LIN {X 0,Y 282.338,Z 475.159,A -85,B 0,C 180,E1 -17007.146,E2 -17007.146} C_VEL
LIN {X 0,Y 282.332,Z 475.749,A -85,B 0,C 180,E1 -17008.574,E2 -17008.574} C_VEL
LIN {X 0,Y 282.332,Z 475.749,A -85,B 0,C 180,E1 -17011.426,E2 -17011.426} C_VEL
LIN {X 0,Y 282.337,Z 475.159,A -85,B 0,C 180,E1 -17012.854,E2 -17012.854} C_VEL
LIN {X 0,Y 282.387,Z 472.707,A -85,B 0,C 180,E1 -17015.713,E2 -17015.713} C_VEL
LIN {X 0,Y 282.677,Z 469.756,A -85,B 0,C 180,E1 -17017.859,E2 -17017.859} C_VEL
LIN {X 0,Y 283.174,Z 465.765,A -85,B 0,C 180,E1 -17020.005,E2 -17020.005} C_VEL
LIN {X 0,Y 283.966,Z 460.633,A -85,B 0,C 180,E1 -17022.144,E2 -17022.144} C_VEL
LIN {X 0,Y 284.95,Z 455.372,A -85,B 0,C 180,E1 -17023.914,E2 -17023.914} C_VEL
LIN {X 0,Y 286.08,Z 449.054,A -85,B 0,C 180,E1 -17025.678,E2 -17025.678} C_VEL
LIN {X 0,Y 287.263,Z 443.105,A -85,B 0,C 180,E1 -17027.073,E2 -17027.073} C_VEL
LIN {X 0,Y 288.401,Z 436.176,A -85,B 0,C 180,E1 -17028.469,E2 -17028.469} C_VEL
LIN {X 0,Y 289.842,Z 427.998,A -85,B 0,C 180,E1 -17029.844,E2 -17029.844} C_VEL
LIN {X 0,Y 291.314,Z 419.49,A -85,B 0,C 180,E1 -17031.03,E2 -17031.03} C_VEL
LIN {X 0,Y 292.62,Z 410.776,A -85,B 0,C 180,E1 -17032.041,E2 -17032.041} C_VEL
LIN {X 0,Y 293.928,Z 401.019,A -85,B 0,C 180,E1 -17032.957,E2 -17032.957} C_VEL
LIN {X 0,Y 295.008,Z 392.229,A -85,B 0,C 180,E1 -17033.611,E2 -17033.611} C_VEL
LIN {X 0,Y 295.879,Z 382.301,A -85,B 0,C 180,E1 -17034.188,E2 -17034.188} C_VEL
LIN {X 0,Y 296.551,Z 372.446,A -85,B 0,C 180,E1 -17034.596,E2 -17034.596} C_VEL
LIN {X 0,Y 297.291,Z 349.624,A -85,B 0,C 180,E1 -17035.184,E2 -17035.184} C_VEL
LIN {X 0,Y 298.183,Z 310.979,A -85,B 0,C 180,E1 -17036.113,E2 -17036.113} C_VEL
LIN {X 0,Y 294.142,Z 288.421,A -85,B 0,C 180,E1 -17037.1,E2 -17037.1} C_VEL
LIN {X 0,Y 290.092,Z 270.616,A -85,B 0,C 180,E1 -17037.994,E2 -17037.994} C_VEL
LIN {X 0,Y 288.061,Z 265.087,A -85,B 0,C 180,E1 -17038.405,E2 -17038.405} C_VEL
LIN {X 0,Y 287.295,Z 260.874,A -85,B 0,C 180,E1 -17040.098,E2 -17040.098} C_VEL
LIN {X 0,Y 285.623,Z 252.564,A -85,B 0,C 180,E1 -17043.784,E2 -17043.784} C_VEL
LIN {X 0,Y 284.361,Z 246.567,A -85,B 0,C 180,E1 -17046.602,E2 -17046.602} C_VEL
LIN {X 0,Y 284.308,Z 246.54,A -85,B 0,C 180,E1 -17049.994,E2 -17049.994} C_VEL
LIN {X 0,Y 284.248,Z 246.575,A -85,B 0,C 180,E1 -17054.19,E2 -17054.19} C_VEL
LIN {X 0,Y 284.274,Z 246.573,A -85,B 0,C 180,E1 -17058.124,E2 -17058.124} C_VEL
LIN {X 0,Y 284.328,Z 246.568,A -85,B 0,C 180,E1 -17062.276,E2 -17062.276} C_VEL
LIN {X 0,Y 284.31,Z 246.548,A -85,B 0,C 180,E1 -17065.35,E2 -17065.35} C_VEL
LIN {X 0,Y 284.295,Z 246.57,A -85,B 0,C 180,E1 -17068.725,E2 -17068.725} C_VEL
LIN {X 0,Y 284.393,Z 246.531,A -85,B 0,C 180,E1 -17072.828,E2 -17072.828} C_VEL
LIN {X 0,Y 284.367,Z 246.56,A -85,B 0,C 180,E1 -17076.706,E2 -17076.706} C_VEL
LIN {X 0,Y 284.383,Z 246.524,A -85,B 0,C 180,E1 -17081.259,E2 -17081.259} C_VEL
LIN {X 0,Y 284.468,Z 246.547,A -85,B 0,C 180,E1 -17085.696,E2 -17085.696} C_VEL
LIN {X 0,Y 284.514,Z 246.504,A -85,B 0,C 180,E1 -17090.042,E2 -17090.042} C_VEL
LIN {X 0,Y 284.653,Z 246.511,A -85,B 0,C 180,E1 -17092.908,E2 -17092.908} C_VEL
LIN {X 0,Y 284.741,Z 246.506,A -85,B 0,C 180,E1 -17097.17,E2 -17097.17} C_VEL
LIN {X 0,Y 284.911,Z 246.454,A -85,B 0,C 180,E1 -17099.999,E2 -17099.999} C_VEL
LIN {X 0,Y 284.743,Z 246.501,A -85,B 0,C 180,E1 -17102.829,E2 -17102.829} C_VEL
LIN {X 0,Y 284.685,Z 246.512,A -85,B 0,C 180,E1 -17107.09,E2 -17107.09} C_VEL
LIN {X 0,Y 284.518,Z 246.504,A -85,B 0,C 180,E1 -17109.956,E2 -17109.956} C_VEL
LIN {X 0,Y 284.48,Z 246.549,A -85,B 0,C 180,E1 -17114.302,E2 -17114.302} C_VEL
LIN {X 0,Y 284.421,Z 246.539,A -85,B 0,C 180,E1 -17117.248,E2 -17117.248} C_VEL
LIN {X 0,Y 284.375,Z 246.533,A -85,B 0,C 180,E1 -17120.242,E2 -17120.242} C_VEL
LIN {X 0,Y 284.334,Z 246.56,A -85,B 0,C 180,E1 -17124.846,E2 -17124.846} C_VEL
LIN {X 0,Y 284.324,Z 246.54,A -85,B 0,C 180,E1 -17128.01,E2 -17128.01} C_VEL
LIN {X 0,Y 284.293,Z 246.573,A -85,B 0,C 180,E1 -17131.274,E2 -17131.274} C_VEL
LIN {X 0,Y 284.359,Z 246.546,A -85,B 0,C 180,E1 -17135.353,E2 -17135.353} C_VEL
LIN {X 0,Y 284.333,Z 246.568,A -85,B 0,C 180,E1 -17138.165,E2 -17138.165} C_VEL
LIN {X 0,Y 284.338,Z 246.558,A -85,B 0,C 180,E1 -17142.14,E2 -17142.14} C_VEL
LIN {X 0,Y 284.293,Z 246.533,A -85,B 0,C 180,E1 -17146.197,E2 -17146.197} C_VEL
LIN {X 0,Y 284.309,Z 246.538,A -85,B 0,C 180,E1 -17150.022,E2 -17150.022} C_VEL
LIN {X 0,Y 284.349,Z 246.546,A -85,B 0,C 180,E1 -17153.617,E2 -17153.617} C_VEL
LIN {X 0,Y 284.304,Z 246.553,A -85,B 0,C 180,E1 -17157.189,E2 -17157.189} C_VEL
LIN {X 0,Y 284.357,Z 246.706,A -85,B 0,C 180,E1 -17160.852,E2 -17160.852} C_VEL
LIN {X 0,Y 284.57,Z 247.628,A -85,B 0,C 180,E1 -17161.125,E2 -17161.125} C_VEL
LIN {X 0,Y 292.692,Z 262.865,A -85,B 0,C 180,E1 -17162.446,E2 -17162.446} C_VEL
LIN {X 0,Y 300.724,Z 274.196,A -85,B 0,C 180,E1 -17163.545,E2 -17163.545} C_VEL
LIN {X 0,Y 308.771,Z 283.256,A -85,B 0,C 180,E1 -17164.599,E2 -17164.599} C_VEL
LIN {X 0,Y 316.781,Z 291.82,A -85,B 0,C 180,E1 -17165.796,E2 -17165.796} C_VEL
LIN {X 0,Y 324.604,Z 299.651,A -85,B 0,C 180,E1 -17167.139,E2 -17167.139} C_VEL
LIN {X 0,Y 333.028,Z 307.638,A -85,B 0,C 180,E1 -17168.762,E2 -17168.762} C_VEL
LIN {X 0,Y 340.838,Z 314.592,A -85,B 0,C 180,E1 -17170.439,E2 -17170.439} C_VEL
LIN {X 0,Y 346.811,Z 319.308,A -85,B 0,C 180,E1 -17171.823,E2 -17171.823} C_VEL
LIN {X 0,Y 352.868,Z 324.611,A -85,B 0,C 180,E1 -17173.385,E2 -17173.385} C_VEL
LIN {X 0,Y 358.666,Z 328.923,A -85,B 0,C 180,E1 -17175.022,E2 -17175.022} C_VEL
LIN {X 0,Y 363.783,Z 333.09,A -85,B 0,C 180,E1 -17176.663,E2 -17176.663} C_VEL
LIN {X 0,Y 368.41,Z 336.029,A -85,B 0,C 180,E1 -17178.317,E2 -17178.317} C_VEL
LIN {X 0,Y 370.505,Z 337.411,A -85,B 0,C 180,E1 -17179.169,E2 -17179.169} C_VEL
LIN {X 0,Y 373.81,Z 340.321,A -85,B 0,C 180,E1 -17180.705,E2 -17180.705} C_VEL
LIN {X 0,Y 376.908,Z 342.491,A -85,B 0,C 180,E1 -17182.387,E2 -17182.387} C_VEL
LIN {X 0,Y 379.747,Z 344.052,A -85,B 0,C 180,E1 -17184.313,E2 -17184.313} C_VEL
LIN {X 0,Y 381.691,Z 344.805,A -85,B 0,C 180,E1 -17186.15,E2 -17186.15} C_VEL
LIN {X 0,Y 382.967,Z 345.365,A -85,B 0,C 180,E1 -17188.16,E2 -17188.16} C_VEL
LIN {X 0,Y 383.351,Z 345.508,A -85,B 0,C 180,E1 -17190,E2 -17190} C_VEL
LIN {X 0,Y 383.05,Z 345.431,A -85,B 0,C 180,E1 -17191.577,E2 -17191.577} C_VEL
LIN {X 0,Y 382.23,Z 344.938,A -85,B 0,C 180,E1 -17193.162,E2 -17193.162} C_VEL
LIN {X 0,Y 380.501,Z 344.425,A -85,B 0,C 180,E1 -17195.024,E2 -17195.024} C_VEL
LIN {X 0,Y 377.946,Z 343.114,A -85,B 0,C 180,E1 -17196.961,E2 -17196.961} C_VEL
LIN {X 0,Y 374.623,Z 340.95,A -85,B 0,C 180,E1 -17198.885,E2 -17198.885} C_VEL
LIN {X 0,Y 371.033,Z 337.887,A -85,B 0,C 180,E1 -17200.604,E2 -17200.604} C_VEL
LIN {X 0,Y 368.789,Z 336.215,A -85,B 0,C 180,E1 -17201.535,E2 -17201.535} C_VEL
LIN {X 0,Y 364.035,Z 333.254,A -85,B 0,C 180,E1 -17203.255,E2 -17203.255} C_VEL
LIN {X 0,Y 359.028,Z 329.244,A -85,B 0,C 180,E1 -17204.863,E2 -17204.863} C_VEL
LIN {X 0,Y 354.264,Z 325.619,A -85,B 0,C 180,E1 -17206.237,E2 -17206.237} C_VEL
LIN {X 0,Y 348.703,Z 321.024,A -85,B 0,C 180,E1 -17207.707,E2 -17207.707} C_VEL
LIN {X 0,Y 341.134,Z 314.874,A -85,B 0,C 180,E1 -17209.492,E2 -17209.492} C_VEL
LIN {X 0,Y 335.412,Z 309.793,A -85,B 0,C 180,E1 -17210.737,E2 -17210.737} C_VEL
LIN {X 0,Y 329.61,Z 304.23,A -85,B 0,C 180,E1 -17211.926,E2 -17211.926} C_VEL
LIN {X 0,Y 323.047,Z 298.018,A -85,B 0,C 180,E1 -17213.151,E2 -17213.151} C_VEL
LIN {X 0,Y 316.393,Z 291.393,A -85,B 0,C 180,E1 -17214.263,E2 -17214.263} C_VEL
LIN {X 0,Y 308.203,Z 282.711,A -85,B 0,C 180,E1 -17215.475,E2 -17215.475} C_VEL
LIN {X 0,Y 299.727,Z 272.881,A -85,B 0,C 180,E1 -17216.585,E2 -17216.585} C_VEL
LIN {X 0,Y 292.26,Z 262.125,A -85,B 0,C 180,E1 -17217.619,E2 -17217.619} C_VEL
LIN {X 0,Y 284.572,Z 247.623,A -85,B 0,C 180,E1 -17218.876,E2 -17218.876} C_VEL
LIN {X 0,Y 284.349,Z 246.627,A -85,B 0,C 180,E1 -17219.19,E2 -17219.19} C_VEL
LIN {X 0,Y 284.302,Z 246.551,A -85,B 0,C 180,E1 -17222.946,E2 -17222.946} C_VEL
LIN {X 0,Y 284.349,Z 246.546,A -85,B 0,C 180,E1 -17226.383,E2 -17226.383} C_VEL
LIN {X 0,Y 284.308,Z 246.538,A -85,B 0,C 180,E1 -17229.994,E2 -17229.994} C_VEL
LIN {X 0,Y 284.29,Z 246.542,A -85,B 0,C 180,E1 -17234.201,E2 -17234.201} C_VEL
LIN {X 0,Y 284.336,Z 246.556,A -85,B 0,C 180,E1 -17238.137,E2 -17238.137} C_VEL
LIN {X 0,Y 284.342,Z 246.568,A -85,B 0,C 180,E1 -17242.272,E2 -17242.272} C_VEL
LIN {X 0,Y 284.321,Z 246.547,A -85,B 0,C 180,E1 -17245.353,E2 -17245.353} C_VEL
LIN {X 0,Y 284.293,Z 246.573,A -85,B 0,C 180,E1 -17248.726,E2 -17248.726} C_VEL
LIN {X 0,Y 284.39,Z 246.53,A -85,B 0,C 180,E1 -17252.829,E2 -17252.829} C_VEL
LIN {X 0,Y 284.331,Z 246.567,A -85,B 0,C 180,E1 -17256.705,E2 -17256.705} C_VEL
LIN {X 0,Y 284.397,Z 246.524,A -85,B 0,C 180,E1 -17261.262,E2 -17261.262} C_VEL
LIN {X 0,Y 284.491,Z 246.545,A -85,B 0,C 180,E1 -17264.46,E2 -17264.46} C_VEL
LIN {X 0,Y 284.486,Z 246.52,A -85,B 0,C 180,E1 -17268.602,E2 -17268.602} C_VEL
LIN {X 0,Y 284.638,Z 246.499,A -85,B 0,C 180,E1 -17271.481,E2 -17271.481} C_VEL
LIN {X 0,Y 284.596,Z 246.533,A -85,B 0,C 180,E1 -17274.332,E2 -17274.332} C_VEL
LIN {X 0,Y 284.854,Z 246.468,A -85,B 0,C 180,E1 -17278.587,E2 -17278.587} C_VEL
LIN {X 0,Y 284.854,Z 246.474,A -85,B 0,C 180,E1 -17281.415,E2 -17281.415} C_VEL
LIN {X 0,Y 284.581,Z 246.533,A -85,B 0,C 180,E1 -17285.67,E2 -17285.67} C_VEL
LIN {X 0,Y 284.615,Z 246.493,A -85,B 0,C 180,E1 -17288.99,E2 -17288.99} C_VEL
LIN {X 0,Y 284.473,Z 246.541,A -85,B 0,C 180,E1 -17292.848,E2 -17292.848} C_VEL
LIN {X 0,Y 284.427,Z 246.546,A -85,B 0,C 180,E1 -17295.772,E2 -17295.772} C_VEL
LIN {X 0,Y 284.383,Z 246.534,A -85,B 0,C 180,E1 -17299.999,E2 -17299.999} C_VEL
LIN {X 0,Y 283.755,Z 246.629,A -85,B 0,C 180,E1 -17301.182,E2 -17301.182} C_VEL
LIN {X 0,Y 280.878,Z 246.995,A -85,B 0,C 180,E1 -17303.107,E2 -17303.107} C_VEL
LIN {X 0,Y 278.419,Z 247.291,A -85,B 0,C 180,E1 -17304.672,E2 -17304.672} C_VEL
LIN {X 0,Y 277.379,Z 247.408,A -85,B 0,C 180,E1 -17305.885,E2 -17305.885} C_VEL
LIN {X 0,Y 277.305,Z 247.414,A -85,B 0,C 180,E1 -17306.296,E2 -17306.296} C_VEL
LIN {X 0,Y 277.273,Z 247.448,A -85,B 0,C 180,E1 -17310.482,E2 -17310.482} C_VEL
LIN {X 0,Y 277.248,Z 247.426,A -85,B 0,C 180,E1 -17313.896,E2 -17313.896} C_VEL
LIN {X 0,Y 277.273,Z 247.446,A -85,B 0,C 180,E1 -17317.469,E2 -17317.469} C_VEL
LIN {X 0,Y 277.212,Z 247.447,A -85,B 0,C 180,E1 -17321.237,E2 -17321.237} C_VEL
LIN {X 0,Y 277.203,Z 247.448,A -85,B 0,C 180,E1 -17325.227,E2 -17325.227} C_VEL
LIN {X 0,Y 277.224,Z 247.421,A -85,B 0,C 180,E1 -17329.513,E2 -17329.513} C_VEL
LIN {X 0,Y 277.351,Z 247.644,A -85,B 0,C 180,E1 -17332.961,E2 -17332.961} C_VEL
LIN {X 0,Y 278.847,Z 254.731,A -85,B 0,C 180,E1 -17336.325,E2 -17336.325} C_VEL
LIN {X 0,Y 280.431,Z 262.591,A -85,B 0,C 180,E1 -17339.919,E2 -17339.919} C_VEL
LIN {X 0,Y 280.834,Z 264.832,A -85,B 0,C 180,E1 -17340.786,E2 -17340.786} C_VEL
LIN {X 0,Y 284.402,Z 274.054,A -85,B 0,C 180,E1 -17341.497,E2 -17341.497} C_VEL
LIN {X 0,Y 289.1,Z 296.203,A -85,B 0,C 180,E1 -17342.605,E2 -17342.605} C_VEL
LIN {X 0,Y 291.885,Z 312.955,A -85,B 0,C 180,E1 -17343.338,E2 -17343.338} C_VEL
LIN {X 0,Y 290.193,Z 370.926,A -85,B 0,C 180,E1 -17344.78,E2 -17344.78} C_VEL
LIN {X 0,Y 289.497,Z 381.234,A -85,B 0,C 180,E1 -17345.195,E2 -17345.195} C_VEL
LIN {X 0,Y 288.564,Z 390.746,A -85,B 0,C 180,E1 -17345.733,E2 -17345.733} C_VEL
LIN {X 0,Y 287.493,Z 399.819,A -85,B 0,C 180,E1 -17346.403,E2 -17346.403} C_VEL
LIN {X 0,Y 286.24,Z 408.95,A -85,B 0,C 180,E1 -17347.25,E2 -17347.25} C_VEL
LIN {X 0,Y 284.929,Z 417.946,A -85,B 0,C 180,E1 -17348.285,E2 -17348.285} C_VEL
LIN {X 0,Y 283.358,Z 426.67,A -85,B 0,C 180,E1 -17349.492,E2 -17349.492} C_VEL
LIN {X 0,Y 281.981,Z 434.062,A -85,B 0,C 180,E1 -17350.717,E2 -17350.717} C_VEL
LIN {X 0,Y 280.72,Z 441.747,A -85,B 0,C 180,E1 -17352.247,E2 -17352.247} C_VEL
LIN {X 0,Y 279.228,Z 448.861,A -85,B 0,C 180,E1 -17353.927,E2 -17353.927} C_VEL
LIN {X 0,Y 278.016,Z 455.178,A -85,B 0,C 180,E1 -17355.731,E2 -17355.731} C_VEL
LIN {X 0,Y 276.987,Z 460.439,A -85,B 0,C 180,E1 -17357.545,E2 -17357.545} C_VEL
LIN {X 0,Y 276.165,Z 465.572,A -85,B 0,C 180,E1 -17359.739,E2 -17359.739} C_VEL
LIN {X 0,Y 275.606,Z 469.562,A -85,B 0,C 180,E1 -17361.938,E2 -17361.938} C_VEL
LIN {X 0,Y 275.254,Z 473.199,A -85,B 0,C 180,E1 -17364.741,E2 -17364.741} C_VEL
LIN {X 0,Y 275.247,Z 474.966,A -85,B 0,C 180,E1 -17367.073,E2 -17367.073} C_VEL
LIN {X 0,Y 275.256,Z 475.557,A -85,B 0,C 180,E1 -17368.537,E2 -17368.537} C_VEL
LIN {X 0,Y 275.256,Z 475.557,A -85,B 0,C 180,E1 -17371.463,E2 -17371.463} C_VEL
LIN {X 0,Y 275.246,Z 474.966,A -85,B 0,C 180,E1 -17372.927,E2 -17372.927} C_VEL
LIN {X 0,Y 275.3,Z 472.514,A -85,B 0,C 180,E1 -17375.861,E2 -17375.861} C_VEL
LIN {X 0,Y 275.606,Z 469.562,A -85,B 0,C 180,E1 -17378.062,E2 -17378.062} C_VEL
LIN {X 0,Y 276.165,Z 465.572,A -85,B 0,C 180,E1 -17380.261,E2 -17380.261} C_VEL
LIN {X 0,Y 276.987,Z 460.439,A -85,B 0,C 180,E1 -17382.455,E2 -17382.455} C_VEL
LIN {X 0,Y 278.014,Z 455.178,A -85,B 0,C 180,E1 -17384.269,E2 -17384.269} C_VEL
LIN {X 0,Y 279.217,Z 448.86,A -85,B 0,C 180,E1 -17386.074,E2 -17386.074} C_VEL
LIN {X 0,Y 280.666,Z 441.91,A -85,B 0,C 180,E1 -17387.718,E2 -17387.718} C_VEL
LIN {X 0,Y 281.662,Z 435.982,A -85,B 0,C 180,E1 -17388.928,E2 -17388.928} C_VEL
LIN {X 0,Y 283.168,Z 427.805,A -85,B 0,C 180,E1 -17390.332,E2 -17390.332} C_VEL
LIN {X 0,Y 284.696,Z 419.297,A -85,B 0,C 180,E1 -17391.543,E2 -17391.543} C_VEL
LIN {X 0,Y 286.054,Z 410.583,A -85,B 0,C 180,E1 -17392.575,E2 -17392.575} C_VEL
LIN {X 0,Y 287.275,Z 401.833,A -85,B 0,C 180,E1 -17393.425,E2 -17393.425} C_VEL
LIN {X 0,Y 288.514,Z 392.036,A -85,B 0,C 180,E1 -17394.176,E2 -17394.176} C_VEL
LIN {X 0,Y 289.425,Z 382.108,A -85,B 0,C 180,E1 -17394.763,E2 -17394.763} C_VEL
LIN {X 0,Y 290.129,Z 372.254,A -85,B 0,C 180,E1 -17395.178,E2 -17395.178} C_VEL
LIN {X 0,Y 290.87,Z 349.431,A -85,B 0,C 180,E1 -17395.78,E2 -17395.78} C_VEL
LIN {X 0,Y 291.736,Z 311.475,A -85,B 0,C 180,E1 -17396.717,E2 -17396.717} C_VEL
LIN {X 0,Y 288.006,Z 290.521,A -85,B 0,C 180,E1 -17397.663,E2 -17397.663} C_VEL
LIN {X 0,Y 284.029,Z 272.943,A -85,B 0,C 180,E1 -17398.575,E2 -17398.575} C_VEL
LIN {X 0,Y 280.833,Z 264.881,A -85,B 0,C 180,E1 -17399.205,E2 -17399.205} C_VEL
LIN {X 0,Y 280.133,Z 261.18,A -85,B 0,C 180,E1 -17400.726,E2 -17400.726} C_VEL
LIN {X 0,Y 278.413,Z 252.737,A -85,B 0,C 180,E1 -17404.608,E2 -17404.608} C_VEL
LIN {X 0,Y 277.328,Z 247.446,A -85,B 0,C 180,E1 -17407.198,E2 -17407.198} C_VEL
LIN {X 0,Y 277.212,Z 247.425,A -85,B 0,C 180,E1 -17411.236,E2 -17411.236} C_VEL
LIN {X 0,Y 277.203,Z 247.445,A -85,B 0,C 180,E1 -17415.226,E2 -17415.226} C_VEL
LIN {X 0,Y 277.224,Z 247.438,A -85,B 0,C 180,E1 -17419.511,E2 -17419.511} C_VEL
LIN {X 0,Y 277.273,Z 247.446,A -85,B 0,C 180,E1 -17422.531,E2 -17422.531} C_VEL
LIN {X 0,Y 277.248,Z 247.426,A -85,B 0,C 180,E1 -17426.104,E2 -17426.104} C_VEL
LIN {X 0,Y 277.263,Z 247.449,A -85,B 0,C 180,E1 -17429.538,E2 -17429.538} C_VEL
LIN {X 0,Y 277.355,Z 247.407,A -85,B 0,C 180,E1 -17432.863,E2 -17432.863} C_VEL
LIN {X 0,Y 277.329,Z 247.436,A -85,B 0,C 180,E1 -17436.079,E2 -17436.079} C_VEL
LIN {X 0,Y 277.333,Z 247.403,A -85,B 0,C 180,E1 -17440.765,E2 -17440.765} C_VEL
LIN {X 0,Y 277.415,Z 247.427,A -85,B 0,C 180,E1 -17445.324,E2 -17445.324} C_VEL
LIN {X 0,Y 277.457,Z 247.384,A -85,B 0,C 180,E1 -17449.786,E2 -17449.786} C_VEL
LIN {X 0,Y 277.611,Z 247.386,A -85,B 0,C 180,E1 -17452.727,E2 -17452.727} C_VEL
LIN {X 0,Y 277.82,Z 247.35,A -85,B 0,C 180,E1 -17458.55,E2 -17458.55} C_VEL
LIN {X 0,Y 277.82,Z 247.344,A -85,B 0,C 180,E1 -17461.449,E2 -17461.449} C_VEL
LIN {X 0,Y 277.64,Z 247.389,A -85,B 0,C 180,E1 -17467.27,E2 -17467.27} C_VEL
LIN {X 0,Y 277.46,Z 247.383,A -85,B 0,C 180,E1 -17470.212,E2 -17470.212} C_VEL
LIN {X 0,Y 277.433,Z 247.428,A -85,B 0,C 180,E1 -17474.673,E2 -17474.673} C_VEL
LIN {X 0,Y 277.34,Z 247.402,A -85,B 0,C 180,E1 -17479.233,E2 -17479.233} C_VEL
LIN {X 0,Y 277.289,Z 247.444,A -85,B 0,C 180,E1 -17484.157,E2 -17484.157} C_VEL
LIN {X 0,Y 277.319,Z 247.41,A -85,B 0,C 180,E1 -17487.503,E2 -17487.503} C_VEL
LIN {X 0,Y 277.269,Z 247.448,A -85,B 0,C 180,E1 -17490.481,E2 -17490.481} C_VEL
LIN {X 0,Y 277.251,Z 247.429,A -85,B 0,C 180,E1 -17493.894,E2 -17493.894} C_VEL
LIN {X 0,Y 277.287,Z 247.446,A -85,B 0,C 180,E1 -17497.465,E2 -17497.465} C_VEL
LIN {X 0,Y 277.261,Z 247.431,A -85,B 0,C 180,E1 -17501.226,E2 -17501.226} C_VEL
LIN {X 0,Y 277.239,Z 247.431,A -85,B 0,C 180,E1 -17505.217,E2 -17505.217} C_VEL
LIN {X 0,Y 277.225,Z 247.408,A -85,B 0,C 180,E1 -17509.51,E2 -17509.51} C_VEL
LIN {X 0,Y 277.285,Z 247.446,A -85,B 0,C 180,E1 -17512.534,E2 -17512.534} C_VEL
LIN {X 0,Y 277.25,Z 247.416,A -85,B 0,C 180,E1 -17516.105,E2 -17516.105} C_VEL
LIN {X 0,Y 277.306,Z 247.573,A -85,B 0,C 180,E1 -17520.072,E2 -17520.072} C_VEL
LIN {X 0,Y 277.558,Z 248.55,A -85,B 0,C 180,E1 -17520.348,E2 -17520.348} C_VEL
LIN {X 0,Y 287.678,Z 267.474,A -85,B 0,C 180,E1 -17522.047,E2 -17522.047} C_VEL
LIN {X 0,Y 296.035,Z 279.257,A -85,B 0,C 180,E1 -17523.224,E2 -17523.224} C_VEL
LIN {X 0,Y 304.941,Z 289.145,A -85,B 0,C 180,E1 -17524.349,E2 -17524.349} C_VEL
LIN {X 0,Y 313.119,Z 297.715,A -85,B 0,C 180,E1 -17525.493,E2 -17525.493} C_VEL
LIN {X 0,Y 322.054,Z 306.384,A -85,B 0,C 180,E1 -17526.937,E2 -17526.937} C_VEL
LIN {X 0,Y 330.86,Z 314.506,A -85,B 0,C 180,E1 -17528.59,E2 -17528.59} C_VEL
LIN {X 0,Y 339.989,Z 322.423,A -85,B 0,C 180,E1 -17530.519,E2 -17530.519} C_VEL
LIN {X 0,Y 346.429,Z 327.558,A -85,B 0,C 180,E1 -17532.016,E2 -17532.016} C_VEL
LIN {X 0,Y 352.732,Z 332.614,A -85,B 0,C 180,E1 -17533.635,E2 -17533.635} C_VEL
LIN {X 0,Y 356.978,Z 335.771,A -85,B 0,C 180,E1 -17534.83,E2 -17534.83} C_VEL
LIN {X 0,Y 362.424,Z 340.053,A -85,B 0,C 180,E1 -17536.544,E2 -17536.544} C_VEL
LIN {X 0,Y 367.359,Z 343.081,A -85,B 0,C 180,E1 -17538.284,E2 -17538.284} C_VEL
LIN {X 0,Y 369.339,Z 344.533,A -85,B 0,C 180,E1 -17539.082,E2 -17539.082} C_VEL
LIN {X 0,Y 373.007,Z 347.551,A -85,B 0,C 180,E1 -17540.763,E2 -17540.763} C_VEL
LIN {X 0,Y 376.178,Z 349.68,A -85,B 0,C 180,E1 -17542.485,E2 -17542.485} C_VEL
LIN {X 0,Y 378.846,Z 351.099,A -85,B 0,C 180,E1 -17544.3,E2 -17544.3} C_VEL
LIN {X 0,Y 380.516,Z 351.761,A -85,B 0,C 180,E1 -17545.826,E2 -17545.826} C_VEL
LIN {X 0,Y 381.686,Z 352.195,A -85,B 0,C 180,E1 -17547.349,E2 -17547.349} C_VEL
LIN {X 0,Y 382.346,Z 352.596,A -85,B 0,C 180,E1 -17548.947,E2 -17548.947} C_VEL
LIN {X 0,Y 382.488,Z 352.539,A -85,B 0,C 180,E1 -17550,E2 -17550} C_VEL
LIN {X 0,Y 382.181,Z 352.479,A -85,B 0,C 180,E1 -17551.581,E2 -17551.581} C_VEL
LIN {X 0,Y 381.093,Z 351.917,A -85,B 0,C 180,E1 -17553.514,E2 -17553.514} C_VEL
LIN {X 0,Y 379.106,Z 351.218,A -85,B 0,C 180,E1 -17555.477,E2 -17555.477} C_VEL
LIN {X 0,Y 376.465,Z 349.809,A -85,B 0,C 180,E1 -17557.348,E2 -17557.348} C_VEL
LIN {X 0,Y 373.181,Z 347.677,A -85,B 0,C 180,E1 -17559.154,E2 -17559.154} C_VEL
LIN {X 0,Y 369.654,Z 344.778,A -85,B 0,C 180,E1 -17560.785,E2 -17560.785} C_VEL
LIN {X 0,Y 366.939,Z 342.836,A -85,B 0,C 180,E1 -17561.871,E2 -17561.871} C_VEL
LIN {X 0,Y 362.246,Z 339.915,A -85,B 0,C 180,E1 -17563.516,E2 -17563.516} C_VEL
LIN {X 0,Y 356.744,Z 335.561,A -85,B 0,C 180,E1 -17565.24,E2 -17565.24} C_VEL
LIN {X 0,Y 349.772,Z 330.397,A -85,B 0,C 180,E1 -17567.136,E2 -17567.136} C_VEL
LIN {X 0,Y 342.455,Z 324.339,A -85,B 0,C 180,E1 -17568.928,E2 -17568.928} C_VEL
LIN {X 0,Y 336.047,Z 318.959,A -85,B 0,C 180,E1 -17570.342,E2 -17570.342} C_VEL
LIN {X 0,Y 328.443,Z 312.315,A -85,B 0,C 180,E1 -17571.883,E2 -17571.883} C_VEL
LIN {X 0,Y 320.06,Z 304.416,A -85,B 0,C 180,E1 -17573.402,E2 -17573.402} C_VEL
LIN {X 0,Y 312.403,Z 296.949,A -85,B 0,C 180,E1 -17574.611,E2 -17574.611} C_VEL
LIN {X 0,Y 303.963,Z 288.179,A -85,B 0,C 180,E1 -17575.775,E2 -17575.775} C_VEL
LIN {X 0,Y 294.557,Z 277.321,A -85,B 0,C 180,E1 -17576.975,E2 -17576.975} C_VEL
LIN {X 0,Y 287.007,Z 266.35,A -85,B 0,C 180,E1 -17578.056,E2 -17578.056} C_VEL
LIN {X 0,Y 277.55,Z 248.559,A -85,B 0,C 180,E1 -17579.65,E2 -17579.65} C_VEL
LIN {X 0,Y 277.302,Z 247.519,A -85,B 0,C 180,E1 -17579.965,E2 -17579.965} C_VEL
LIN {X 0,Y 277.25,Z 247.416,A -85,B 0,C 180,E1 -17583.895,E2 -17583.895} C_VEL
LIN {X 0,Y 277.285,Z 247.446,A -85,B 0,C 180,E1 -17587.466,E2 -17587.466} C_VEL
LIN {X 0,Y 277.214,Z 247.401,A -85,B 0,C 180,E1 -17591.235,E2 -17591.235} C_VEL
LIN {X 0,Y 277.243,Z 247.439,A -85,B 0,C 180,E1 -17595.217,E2 -17595.217} C_VEL
LIN {X 0,Y 277.292,Z 247.426,A -85,B 0,C 180,E1 -17599.495,E2 -17599.495} C_VEL
LIN {X 0,Y 277.287,Z 247.446,A -85,B 0,C 180,E1 -17602.535,E2 -17602.535} C_VEL
LIN {X 0,Y 277.251,Z 247.429,A -85,B 0,C 180,E1 -17606.106,E2 -17606.106} C_VEL
LIN {X 0,Y 277.259,Z 247.449,A -85,B 0,C 180,E1 -17609.539,E2 -17609.539} C_VEL
LIN {X 0,Y 277.352,Z 247.406,A -85,B 0,C 180,E1 -17612.864,E2 -17612.864} C_VEL
LIN {X 0,Y 277.295,Z 247.445,A -85,B 0,C 180,E1 -17616.077,E2 -17616.077} C_VEL
LIN {X 0,Y 277.34,Z 247.402,A -85,B 0,C 180,E1 -17620.767,E2 -17620.767} C_VEL
LIN {X 0,Y 277.433,Z 247.428,A -85,B 0,C 180,E1 -17625.327,E2 -17625.327} C_VEL
LIN {X 0,Y 277.46,Z 247.383,A -85,B 0,C 180,E1 -17629.788,E2 -17629.788} C_VEL
LIN {X 0,Y 277.64,Z 247.389,A -85,B 0,C 180,E1 -17632.73,E2 -17632.73} C_VEL
LIN {X 0,Y 277.82,Z 247.344,A -85,B 0,C 180,E1 -17638.551,E2 -17638.551} C_VEL
LIN {X 0,Y 277.82,Z 247.35,A -85,B 0,C 180,E1 -17641.45,E2 -17641.45} C_VEL
LIN {X 0,Y 277.611,Z 247.386,A -85,B 0,C 180,E1 -17647.273,E2 -17647.273} C_VEL
LIN {X 0,Y 277.457,Z 247.384,A -85,B 0,C 180,E1 -17650.214,E2 -17650.214} C_VEL
LIN {X 0,Y 277.415,Z 247.427,A -85,B 0,C 180,E1 -17654.676,E2 -17654.676} C_VEL
LIN {X 0,Y 277.333,Z 247.403,A -85,B 0,C 180,E1 -17659.235,E2 -17659.235} C_VEL
LIN {X 0,Y 277.329,Z 247.436,A -85,B 0,C 180,E1 -17663.921,E2 -17663.921} C_VEL
LIN {X 0,Y 277.305,Z 247.414,A -85,B 0,C 180,E1 -17666.296,E2 -17666.296} C_VEL
LIN {X 0,Y 276.644,Z 247.5,A -85,B 0,C 180,E1 -17667.508,E2 -17667.508} C_VEL
LIN {X 0,Y 273.728,Z 247.885,A -85,B 0,C 180,E1 -17669.48,E2 -17669.48} C_VEL
LIN {X 0,Y 271.265,Z 248.194,A -85,B 0,C 180,E1 -17671.083,E2 -17671.083} C_VEL
LIN {X 0,Y 270.243,Z 248.311,A -85,B 0,C 180,E1 -17672.328,E2 -17672.328} C_VEL
LIN {X 0,Y 270.179,Z 248.312,A -85,B 0,C 180,E1 -17672.749,E2 -17672.749} C_VEL
LIN {X 0,Y 270.229,Z 248.323,A -85,B 0,C 180,E1 -17676.74,E2 -17676.74} C_VEL
LIN {X 0,Y 270.171,Z 248.321,A -85,B 0,C 180,E1 -17681.029,E2 -17681.029} C_VEL
LIN {X 0,Y 270.154,Z 248.327,A -85,B 0,C 180,E1 -17685.381,E2 -17685.381} C_VEL
LIN {X 0,Y 270.176,Z 248.298,A -85,B 0,C 180,E1 -17689.435,E2 -17689.435} C_VEL
LIN {X 0,Y 270.284,Z 248.51,A -85,B 0,C 180,E1 -17692.335,E2 -17692.335} C_VEL
LIN {X 0,Y 271.788,Z 255.647,A -85,B 0,C 180,E1 -17695.841,E2 -17695.841} C_VEL
LIN {X 0,Y 273.486,Z 264.006,A -85,B 0,C 180,E1 -17699.764,E2 -17699.764} C_VEL
LIN {X 0,Y 273.78,Z 265.178,A -85,B 0,C 180,E1 -17700.007,E2 -17700.007} C_VEL
LIN {X 0,Y 278.471,Z 276.628,A -85,B 0,C 180,E1 -17700.912,E2 -17700.912} C_VEL
LIN {X 0,Y 283.548,Z 301.422,A -85,B 0,C 180,E1 -17702.173,E2 -17702.173} C_VEL
LIN {X 0,Y 285.508,Z 313.952,A -85,B 0,C 180,E1 -17702.726,E2 -17702.726} C_VEL
LIN {X 0,Y 283.783,Z 370.74,A -85,B 0,C 180,E1 -17704.169,E2 -17704.169} C_VEL
LIN {X 0,Y 283.055,Z 381.041,A -85,B 0,C 180,E1 -17704.591,E2 -17704.591} C_VEL
LIN {X 0,Y 282.119,Z 390.554,A -85,B 0,C 180,E1 -17705.141,E2 -17705.141} C_VEL
LIN {X 0,Y 281.007,Z 399.626,A -85,B 0,C 180,E1 -17705.824,E2 -17705.824} C_VEL
LIN {X 0,Y 279.702,Z 408.757,A -85,B 0,C 180,E1 -17706.688,E2 -17706.688} C_VEL
LIN {X 0,Y 278.331,Z 417.753,A -85,B 0,C 180,E1 -17707.743,E2 -17707.743} C_VEL
LIN {X 0,Y 276.694,Z 426.477,A -85,B 0,C 180,E1 -17708.975,E2 -17708.975} C_VEL
LIN {X 0,Y 275.282,Z 433.869,A -85,B 0,C 180,E1 -17710.228,E2 -17710.228} C_VEL
LIN {X 0,Y 273.99,Z 440.886,A -85,B 0,C 180,E1 -17711.638,E2 -17711.638} C_VEL
LIN {X 0,Y 272.711,Z 447.292,A -85,B 0,C 180,E1 -17713.147,E2 -17713.147} C_VEL
LIN {X 0,Y 271.386,Z 453.829,A -85,B 0,C 180,E1 -17714.991,E2 -17714.991} C_VEL
LIN {X 0,Y 270.417,Z 458.329,A -85,B 0,C 180,E1 -17716.473,E2 -17716.473} C_VEL
LIN {X 0,Y 269.414,Z 463.823,A -85,B 0,C 180,E1 -17718.718,E2 -17718.718} C_VEL
LIN {X 0,Y 268.707,Z 468.15,A -85,B 0,C 180,E1 -17720.971,E2 -17720.971} C_VEL
LIN {X 0,Y 268.419,Z 470.52,A -85,B 0,C 180,E1 -17722.478,E2 -17722.478} C_VEL
LIN {X 0,Y 268.167,Z 473.174,A -85,B 0,C 180,E1 -17724.809,E2 -17724.809} C_VEL
LIN {X 0,Y 268.158,Z 474.773,A -85,B 0,C 180,E1 -17726.995,E2 -17726.995} C_VEL
LIN {X 0,Y 268.182,Z 475.365,A -85,B 0,C 180,E1 -17728.498,E2 -17728.498} C_VEL
LIN {X 0,Y 268.182,Z 475.365,A -85,B 0,C 180,E1 -17731.502,E2 -17731.502} C_VEL
LIN {X 0,Y 268.157,Z 474.773,A -85,B 0,C 180,E1 -17733.005,E2 -17733.005} C_VEL
LIN {X 0,Y 268.225,Z 472.321,A -85,B 0,C 180,E1 -17736.016,E2 -17736.016} C_VEL
LIN {X 0,Y 268.548,Z 469.368,A -85,B 0,C 180,E1 -17738.276,E2 -17738.276} C_VEL
LIN {X 0,Y 269.154,Z 465.378,A -85,B 0,C 180,E1 -17740.532,E2 -17740.532} C_VEL
LIN {X 0,Y 270.027,Z 460.245,A -85,B 0,C 180,E1 -17742.781,E2 -17742.781} C_VEL
LIN {X 0,Y 271.109,Z 454.984,A -85,B 0,C 180,E1 -17744.64,E2 -17744.64} C_VEL
LIN {X 0,Y 272.381,Z 448.667,A -85,B 0,C 180,E1 -17746.488,E2 -17746.488} C_VEL
LIN {X 0,Y 273.661,Z 442.718,A -85,B 0,C 180,E1 -17747.949,E2 -17747.949} C_VEL
LIN {X 0,Y 274.93,Z 435.789,A -85,B 0,C 180,E1 -17749.409,E2 -17749.409} C_VEL
LIN {X 0,Y 276.499,Z 427.612,A -85,B 0,C 180,E1 -17750.845,E2 -17750.845} C_VEL
LIN {X 0,Y 278.088,Z 419.104,A -85,B 0,C 180,E1 -17752.082,E2 -17752.082} C_VEL
LIN {X 0,Y 279.506,Z 410.39,A -85,B 0,C 180,E1 -17753.134,E2 -17753.134} C_VEL
LIN {X 0,Y 280.776,Z 401.641,A -85,B 0,C 180,E1 -17754.001,E2 -17754.001} C_VEL
LIN {X 0,Y 282.045,Z 391.843,A -85,B 0,C 180,E1 -17754.767,E2 -17754.767} C_VEL
LIN {X 0,Y 283.002,Z 381.916,A -85,B 0,C 180,E1 -17755.365,E2 -17755.365} C_VEL
LIN {X 0,Y 283.722,Z 372.061,A -85,B 0,C 180,E1 -17755.787,E2 -17755.787} C_VEL
LIN {X 0,Y 284.524,Z 348.19,A -85,B 0,C 180,E1 -17756.428,E2 -17756.428} C_VEL
LIN {X 0,Y 285.401,Z 312.621,A -85,B 0,C 180,E1 -17757.322,E2 -17757.322} C_VEL
LIN {X 0,Y 281.498,Z 290.788,A -85,B 0,C 180,E1 -17758.347,E2 -17758.347} C_VEL
LIN {X 0,Y 278.14,Z 275.732,A -85,B 0,C 180,E1 -17759.152,E2 -17759.152} C_VEL
LIN {X 0,Y 273.668,Z 264.892,A -85,B 0,C 180,E1 -17760.02,E2 -17760.02} C_VEL
LIN {X 0,Y 273.481,Z 264.039,A -85,B 0,C 180,E1 -17760.231,E2 -17760.231} C_VEL
LIN {X 0,Y 271.813,Z 255.624,A -85,B 0,C 180,E1 -17764.167,E2 -17764.167} C_VEL
LIN {X 0,Y 270.256,Z 248.332,A -85,B 0,C 180,E1 -17767.847,E2 -17767.847} C_VEL
LIN {X 0,Y 270.174,Z 248.321,A -85,B 0,C 180,E1 -17772.558,E2 -17772.558} C_VEL
LIN {X 0,Y 270.167,Z 248.329,A -85,B 0,C 180,E1 -17776.75,E2 -17776.75} C_VEL
LIN {X 0,Y 270.176,Z 248.316,A -85,B 0,C 180,E1 -17779.434,E2 -17779.434} C_VEL
LIN {X 0,Y 270.244,Z 248.317,A -85,B 0,C 180,E1 -17783.725,E2 -17783.725} C_VEL
LIN {X 0,Y 270.204,Z 248.308,A -85,B 0,C 180,E1 -17786.892,E2 -17786.892} C_VEL
LIN {X 0,Y 270.196,Z 248.325,A -85,B 0,C 180,E1 -17790.382,E2 -17790.382} C_VEL
LIN {X 0,Y 270.261,Z 248.291,A -85,B 0,C 180,E1 -17793.763,E2 -17793.763} C_VEL
LIN {X 0,Y 270.233,Z 248.323,A -85,B 0,C 180,E1 -17797.038,E2 -17797.038} C_VEL
LIN {X 0,Y 270.28,Z 248.286,A -85,B 0,C 180,E1 -17800.242,E2 -17800.242} C_VEL
LIN {X 0,Y 270.374,Z 248.3,A -85,B 0,C 180,E1 -17804.933,E2 -17804.933} C_VEL
LIN {X 0,Y 270.41,Z 248.263,A -85,B 0,C 180,E1 -17809.517,E2 -17809.517} C_VEL
LIN {X 0,Y 270.57,Z 248.261,A -85,B 0,C 180,E1 -17812.537,E2 -17812.537} C_VEL
LIN {X 0,Y 270.786,Z 248.225,A -85,B 0,C 180,E1 -17818.512,E2 -17818.512} C_VEL
LIN {X 0,Y 270.786,Z 248.219,A -85,B 0,C 180,E1 -17821.486,E2 -17821.486} C_VEL
LIN {X 0,Y 270.598,Z 248.264,A -85,B 0,C 180,E1 -17827.461,E2 -17827.461} C_VEL
LIN {X 0,Y 270.412,Z 248.261,A -85,B 0,C 180,E1 -17830.481,E2 -17830.481} C_VEL
LIN {X 0,Y 270.402,Z 248.301,A -85,B 0,C 180,E1 -17835.064,E2 -17835.064} C_VEL
LIN {X 0,Y 270.298,Z 248.28,A -85,B 0,C 180,E1 -17839.755,E2 -17839.755} C_VEL
LIN {X 0,Y 270.235,Z 248.318,A -85,B 0,C 180,E1 -17844.588,E2 -17844.588} C_VEL
LIN {X 0,Y 270.267,Z 248.289,A -85,B 0,C 180,E1 -17847.908,E2 -17847.908} C_VEL
LIN {X 0,Y 270.182,Z 248.331,A -85,B 0,C 180,E1 -17851.347,E2 -17851.347} C_VEL
LIN {X 0,Y 270.213,Z 248.304,A -85,B 0,C 180,E1 -17854.903,E2 -17854.903} C_VEL
LIN {X 0,Y 270.219,Z 248.323,A -85,B 0,C 180,E1 -17858.716,E2 -17858.716} C_VEL
LIN {X 0,Y 270.22,Z 248.322,A -85,B 0,C 180,E1 -17862.548,E2 -17862.548} C_VEL
LIN {X 0,Y 270.186,Z 248.279,A -85,B 0,C 180,E1 -17866.745,E2 -17866.745} C_VEL
LIN {X 0,Y 270.209,Z 248.324,A -85,B 0,C 180,E1 -17871.375,E2 -17871.375} C_VEL
LIN {X 0,Y 270.212,Z 248.289,A -85,B 0,C 180,E1 -17875.096,E2 -17875.096} C_VEL
LIN {X 0,Y 270.248,Z 248.542,A -85,B 0,C 180,E1 -17879.292,E2 -17879.292} C_VEL
LIN {X 0,Y 270.53,Z 249.639,A -85,B 0,C 180,E1 -17879.534,E2 -17879.534} C_VEL
LIN {X 0,Y 282.824,Z 272.311,A -85,B 0,C 180,E1 -17881.657,E2 -17881.657} C_VEL
LIN {X 0,Y 291.273,Z 284.221,A -85,B 0,C 180,E1 -17882.881,E2 -17882.881} C_VEL
LIN {X 0,Y 300.227,Z 294.168,A -85,B 0,C 180,E1 -17884.02,E2 -17884.02} C_VEL
LIN {X 0,Y 307.234,Z 301.324,A -85,B 0,C 180,E1 -17884.917,E2 -17884.917} C_VEL
LIN {X 0,Y 313.893,Z 307.826,A -85,B 0,C 180,E1 -17885.871,E2 -17885.871} C_VEL
LIN {X 0,Y 321.78,Z 315.113,A -85,B 0,C 180,E1 -17887.148,E2 -17887.148} C_VEL
LIN {X 0,Y 329.962,Z 322.469,A -85,B 0,C 180,E1 -17888.674,E2 -17888.674} C_VEL
LIN {X 0,Y 338.441,Z 329.612,A -85,B 0,C 180,E1 -17890.442,E2 -17890.442} C_VEL
LIN {X 0,Y 343.949,Z 333.947,A -85,B 0,C 180,E1 -17891.702,E2 -17891.702} C_VEL
LIN {X 0,Y 349.913,Z 338.662,A -85,B 0,C 180,E1 -17893.181,E2 -17893.181} C_VEL
LIN {X 0,Y 355.219,Z 342.572,A -85,B 0,C 180,E1 -17894.623,E2 -17894.623} C_VEL
LIN {X 0,Y 361.118,Z 347.048,A -85,B 0,C 180,E1 -17896.441,E2 -17896.441} C_VEL
LIN {X 0,Y 366.164,Z 350.063,A -85,B 0,C 180,E1 -17898.198,E2 -17898.198} C_VEL
LIN {X 0,Y 369.109,Z 352.416,A -85,B 0,C 180,E1 -17899.391,E2 -17899.391} C_VEL
LIN {X 0,Y 373.006,Z 355.358,A -85,B 0,C 180,E1 -17901.232,E2 -17901.232} C_VEL
LIN {X 0,Y 376.419,Z 357.386,A -85,B 0,C 180,E1 -17903.208,E2 -17903.208} C_VEL
LIN {X 0,Y 378.71,Z 358.506,A -85,B 0,C 180,E1 -17904.946,E2 -17904.946} C_VEL
LIN {X 0,Y 380.674,Z 359.126,A -85,B 0,C 180,E1 -17907.083,E2 -17907.083} C_VEL
LIN {X 0,Y 381.48,Z 359.642,A -85,B 0,C 180,E1 -17908.944,E2 -17908.944} C_VEL
LIN {X 0,Y 381.624,Z 359.577,A -85,B 0,C 180,E1 -17910,E2 -17910} C_VEL
LIN {X 0,Y 381.313,Z 359.519,A -85,B 0,C 180,E1 -17911.584,E2 -17911.584} C_VEL
LIN {X 0,Y 380.223,Z 358.936,A -85,B 0,C 180,E1 -17913.517,E2 -17913.517} C_VEL
LIN {X 0,Y 378.214,Z 358.268,A -85,B 0,C 180,E1 -17915.49,E2 -17915.49} C_VEL
LIN {X 0,Y 375.564,Z 356.906,A -85,B 0,C 180,E1 -17917.348,E2 -17917.348} C_VEL
LIN {X 0,Y 372.201,Z 354.806,A -85,B 0,C 180,E1 -17919.178,E2 -17919.178} C_VEL
LIN {X 0,Y 368.461,Z 351.87,A -85,B 0,C 180,E1 -17920.883,E2 -17920.883} C_VEL
LIN {X 0,Y 366.019,Z 349.982,A -85,B 0,C 180,E1 -17921.856,E2 -17921.856} C_VEL
LIN {X 0,Y 361.119,Z 347.043,A -85,B 0,C 180,E1 -17923.559,E2 -17923.559} C_VEL
LIN {X 0,Y 355.429,Z 342.731,A -85,B 0,C 180,E1 -17925.317,E2 -17925.317} C_VEL
LIN {X 0,Y 348.215,Z 337.421,A -85,B 0,C 180,E1 -17927.249,E2 -17927.249} C_VEL
LIN {X 0,Y 342.464,Z 332.596,A -85,B 0,C 180,E1 -17928.66,E2 -17928.66} C_VEL
LIN {X 0,Y 335.483,Z 327.228,A -85,B 0,C 180,E1 -17930.193,E2 -17930.193} C_VEL
LIN {X 0,Y 327.646,Z 320.511,A -85,B 0,C 180,E1 -17931.774,E2 -17931.774} C_VEL
LIN {X 0,Y 318.88,Z 312.572,A -85,B 0,C 180,E1 -17933.336,E2 -17933.336} C_VEL
LIN {X 0,Y 309.767,Z 303.993,A -85,B 0,C 180,E1 -17934.728,E2 -17934.728} C_VEL
LIN {X 0,Y 300.893,Z 294.901,A -85,B 0,C 180,E1 -17935.898,E2 -17935.898} C_VEL
LIN {X 0,Y 290.789,Z 283.583,A -85,B 0,C 180,E1 -17937.185,E2 -17937.185} C_VEL
LIN {X 0,Y 282.328,Z 271.548,A -85,B 0,C 180,E1 -17938.419,E2 -17938.419} C_VEL
LIN {X 0,Y 271.16,Z 251.042,A -85,B 0,C 180,E1 -17940.33,E2 -17940.33} C_VEL
LIN {X 0,Y 270.369,Z 249.024,A -85,B 0,C 180,E1 -17940.563,E2 -17940.563} C_VEL
LIN {X 0,Y 270.204,Z 248.375,A -85,B 0,C 180,E1 -17940.872,E2 -17940.872} C_VEL
LIN {X 0,Y 270.212,Z 248.289,A -85,B 0,C 180,E1 -17944.904,E2 -17944.904} C_VEL
LIN {X 0,Y 270.219,Z 248.32,A -85,B 0,C 180,E1 -17948.717,E2 -17948.717} C_VEL
LIN {X 0,Y 270.186,Z 248.279,A -85,B 0,C 180,E1 -17953.255,E2 -17953.255} C_VEL
LIN {X 0,Y 270.22,Z 248.322,A -85,B 0,C 180,E1 -17957.452,E2 -17957.452} C_VEL
LIN {X 0,Y 270.242,Z 248.32,A -85,B 0,C 180,E1 -17961.381,E2 -17961.381} C_VEL
LIN {X 0,Y 270.213,Z 248.304,A -85,B 0,C 180,E1 -17965.097,E2 -17965.097} C_VEL
LIN {X 0,Y 270.198,Z 248.329,A -85,B 0,C 180,E1 -17969.131,E2 -17969.131} C_VEL
LIN {X 0,Y 270.26,Z 248.29,A -85,B 0,C 180,E1 -17972.147,E2 -17972.147} C_VEL
LIN {X 0,Y 270.235,Z 248.319,A -85,B 0,C 180,E1 -17975.539,E2 -17975.539} C_VEL
LIN {X 0,Y 270.298,Z 248.28,A -85,B 0,C 180,E1 -17980.245,E2 -17980.245} C_VEL
LIN {X 0,Y 270.402,Z 248.301,A -85,B 0,C 180,E1 -17984.936,E2 -17984.936} C_VEL
LIN {X 0,Y 270.412,Z 248.261,A -85,B 0,C 180,E1 -17989.519,E2 -17989.519} C_VEL
LIN {X 0,Y 270.598,Z 248.264,A -85,B 0,C 180,E1 -17992.539,E2 -17992.539} C_VEL
LIN {X 0,Y 270.786,Z 248.219,A -85,B 0,C 180,E1 -17998.514,E2 -17998.514} C_VEL
LIN {X 0,Y 270.786,Z 248.225,A -85,B 0,C 180,E1 -18001.488,E2 -18001.488} C_VEL
LIN {X 0,Y 270.57,Z 248.261,A -85,B 0,C 180,E1 -18007.463,E2 -18007.463} C_VEL
LIN {X 0,Y 270.41,Z 248.263,A -85,B 0,C 180,E1 -18010.483,E2 -18010.483} C_VEL
LIN {X 0,Y 270.374,Z 248.3,A -85,B 0,C 180,E1 -18015.067,E2 -18015.067} C_VEL
LIN {X 0,Y 270.28,Z 248.286,A -85,B 0,C 180,E1 -18019.758,E2 -18019.758} C_VEL
LIN {X 0,Y 270.275,Z 248.306,A -85,B 0,C 180,E1 -18024.586,E2 -18024.586} C_VEL
LIN {X 0,Y 270.27,Z 248.294,A -85,B 0,C 180,E1 -18027.91,E2 -18027.91} C_VEL
LIN {X 0,Y 270.185,Z 248.328,A -85,B 0,C 180,E1 -18031.349,E2 -18031.349} C_VEL
LIN {X 0,Y 270.179,Z 248.312,A -85,B 0,C 180,E1 -18032.749,E2 -18032.749} C_VEL
LIN {X 0,Y 269.566,Z 248.388,A -85,B 0,C 180,E1 -18033.994,E2 -18033.994} C_VEL
LIN {X 0,Y 266.731,Z 248.753,A -85,B 0,C 180,E1 -18036.023,E2 -18036.023} C_VEL
LIN {X 0,Y 264.28,Z 249.065,A -85,B 0,C 180,E1 -18037.672,E2 -18037.672} C_VEL
LIN {X 0,Y 263.209,Z 249.187,A -85,B 0,C 180,E1 -18038.951,E2 -18038.951} C_VEL
LIN {X 0,Y 263.114,Z 249.196,A -85,B 0,C 180,E1 -18039.385,E2 -18039.385} C_VEL
LIN {X 0,Y 263.126,Z 249.207,A -85,B 0,C 180,E1 -18041.894,E2 -18041.894} C_VEL
LIN {X 0,Y 263.126,Z 249.21,A -85,B 0,C 180,E1 -18046.151,E2 -18046.151} C_VEL
LIN {X 0,Y 263.108,Z 249.179,A -85,B 0,C 180,E1 -18050.128,E2 -18050.128} C_VEL
LIN {X 0,Y 263.216,Z 249.317,A -85,B 0,C 180,E1 -18051.636,E2 -18051.636} C_VEL
LIN {X 0,Y 264.779,Z 256.641,A -85,B 0,C 180,E1 -18055.37,E2 -18055.37} C_VEL
LIN {X 0,Y 266.296,Z 264.192,A -85,B 0,C 180,E1 -18058.979,E2 -18058.979} C_VEL
LIN {X 0,Y 267.656,Z 267.6,A -85,B 0,C 180,E1 -18059.351,E2 -18059.351} C_VEL
LIN {X 0,Y 272.536,Z 279.176,A -85,B 0,C 180,E1 -18060.296,E2 -18060.296} C_VEL
LIN {X 0,Y 277.456,Z 303.571,A -85,B 0,C 180,E1 -18061.574,E2 -18061.574} C_VEL
LIN {X 0,Y 279.176,Z 314.792,A -85,B 0,C 180,E1 -18062.084,E2 -18062.084} C_VEL
LIN {X 0,Y 277.421,Z 370.554,A -85,B 0,C 180,E1 -18063.531,E2 -18063.531} C_VEL
LIN {X 0,Y 276.644,Z 380.848,A -85,B 0,C 180,E1 -18063.959,E2 -18063.959} C_VEL
LIN {X 0,Y 275.702,Z 390.361,A -85,B 0,C 180,E1 -18064.522,E2 -18064.522} C_VEL
LIN {X 0,Y 274.544,Z 399.433,A -85,B 0,C 180,E1 -18065.217,E2 -18065.217} C_VEL
LIN {X 0,Y 273.2,Z 408.564,A -85,B 0,C 180,E1 -18066.099,E2 -18066.099} C_VEL
LIN {X 0,Y 271.748,Z 417.56,A -85,B 0,C 180,E1 -18067.174,E2 -18067.174} C_VEL
LIN {X 0,Y 270.089,Z 426.284,A -85,B 0,C 180,E1 -18068.436,E2 -18068.436} C_VEL
LIN {X 0,Y 268.581,Z 433.676,A -85,B 0,C 180,E1 -18069.714,E2 -18069.714} C_VEL
LIN {X 0,Y 267.086,Z 441.39,A -85,B 0,C 180,E1 -18071.316,E2 -18071.316} C_VEL
LIN {X 0,Y 265.917,Z 447.099,A -85,B 0,C 180,E1 -18072.703,E2 -18072.703} C_VEL
LIN {X 0,Y 264.507,Z 453.636,A -85,B 0,C 180,E1 -18074.591,E2 -18074.591} C_VEL
LIN {X 0,Y 263.507,Z 458.136,A -85,B 0,C 180,E1 -18076.111,E2 -18076.111} C_VEL
LIN {X 0,Y 262.419,Z 463.63,A -85,B 0,C 180,E1 -18078.413,E2 -18078.413} C_VEL
LIN {X 0,Y 261.687,Z 467.957,A -85,B 0,C 180,E1 -18080.727,E2 -18080.727} C_VEL
LIN {X 0,Y 261.353,Z 470.326,A -85,B 0,C 180,E1 -18082.273,E2 -18082.273} C_VEL
LIN {X 0,Y 261.087,Z 473.132,A -85,B 0,C 180,E1 -18084.865,E2 -18084.865} C_VEL
LIN {X 0,Y 261.054,Z 474.58,A -85,B 0,C 180,E1 -18086.914,E2 -18086.914} C_VEL
LIN {X 0,Y 261.088,Z 475.172,A -85,B 0,C 180,E1 -18088.458,E2 -18088.458} C_VEL
LIN {X 0,Y 261.088,Z 475.172,A -85,B 0,C 180,E1 -18091.542,E2 -18091.542} C_VEL
LIN {X 0,Y 261.052,Z 474.58,A -85,B 0,C 180,E1 -18093.086,E2 -18093.086} C_VEL
LIN {X 0,Y 261.151,Z 472.128,A -85,B 0,C 180,E1 -18096.18,E2 -18096.18} C_VEL
LIN {X 0,Y 261.511,Z 469.175,A -85,B 0,C 180,E1 -18098.5,E2 -18098.5} C_VEL
LIN {X 0,Y 262.131,Z 465.184,A -85,B 0,C 180,E1 -18100.817,E2 -18100.817} C_VEL
LIN {X 0,Y 263.085,Z 460.052,A -85,B 0,C 180,E1 -18103.124,E2 -18103.124} C_VEL
LIN {X 0,Y 264.228,Z 454.791,A -85,B 0,C 180,E1 -18105.03,E2 -18105.03} C_VEL
LIN {X 0,Y 265.567,Z 448.474,A -85,B 0,C 180,E1 -18106.924,E2 -18106.924} C_VEL
LIN {X 0,Y 266.865,Z 442.524,A -85,B 0,C 180,E1 -18108.423,E2 -18108.423} C_VEL
LIN {X 0,Y 268.222,Z 435.596,A -85,B 0,C 180,E1 -18109.915,E2 -18109.915} C_VEL
LIN {X 0,Y 269.868,Z 427.419,A -85,B 0,C 180,E1 -18111.382,E2 -18111.382} C_VEL
LIN {X 0,Y 271.503,Z 418.911,A -85,B 0,C 180,E1 -18112.647,E2 -18112.647} C_VEL
LIN {X 0,Y 272.991,Z 410.197,A -85,B 0,C 180,E1 -18113.719,E2 -18113.719} C_VEL
LIN {X 0,Y 274.313,Z 401.448,A -85,B 0,C 180,E1 -18114.603,E2 -18114.603} C_VEL
LIN {X 0,Y 275.593,Z 391.65,A -85,B 0,C 180,E1 -18115.388,E2 -18115.388} C_VEL
LIN {X 0,Y 276.588,Z 381.723,A -85,B 0,C 180,E1 -18115.996,E2 -18115.996} C_VEL
LIN {X 0,Y 277.355,Z 371.869,A -85,B 0,C 180,E1 -18116.425,E2 -18116.425} C_VEL
LIN {X 0,Y 278.207,Z 347.703,A -85,B 0,C 180,E1 -18117.084,E2 -18117.084} C_VEL
LIN {X 0,Y 279.117,Z 313.756,A -85,B 0,C 180,E1 -18117.952,E2 -18117.952} C_VEL
LIN {X 0,Y 275.332,Z 292.465,A -85,B 0,C 180,E1 -18118.987,E2 -18118.987} C_VEL
LIN {X 0,Y 272.218,Z 278.332,A -85,B 0,C 180,E1 -18119.767,E2 -18119.767} C_VEL
LIN {X 0,Y 266.4,Z 264.617,A -85,B 0,C 180,E1 -18120.934,E2 -18120.934} C_VEL
LIN {X 0,Y 266.159,Z 263.447,A -85,B 0,C 180,E1 -18121.295,E2 -18121.295} C_VEL
LIN {X 0,Y 264.586,Z 255.697,A -85,B 0,C 180,E1 -18125.097,E2 -18125.097} C_VEL
LIN {X 0,Y 263.202,Z 249.222,A -85,B 0,C 180,E1 -18128.486,E2 -18128.486} C_VEL
LIN {X 0,Y 263.126,Z 249.186,A -85,B 0,C 180,E1 -18131.893,E2 -18131.893} C_VEL
LIN {X 0,Y 263.107,Z 249.202,A -85,B 0,C 180,E1 -18136.154,E2 -18136.154} C_VEL
LIN {X 0,Y 263.107,Z 249.195,A -85,B 0,C 180,E1 -18140.127,E2 -18140.127} C_VEL
LIN {X 0,Y 263.177,Z 249.195,A -85,B 0,C 180,E1 -18144.019,E2 -18144.019} C_VEL
LIN {X 0,Y 263.134,Z 249.197,A -85,B 0,C 180,E1 -18147.711,E2 -18147.711} C_VEL
LIN {X 0,Y 263.197,Z 249.178,A -85,B 0,C 180,E1 -18151.785,E2 -18151.785} C_VEL
LIN {X 0,Y 263.227,Z 249.182,A -85,B 0,C 180,E1 -18155.2,E2 -18155.2} C_VEL
LIN {X 0,Y 263.258,Z 249.167,A -85,B 0,C 180,E1 -18159.692,E2 -18159.692} C_VEL
LIN {X 0,Y 263.315,Z 249.177,A -85,B 0,C 180,E1 -18164.519,E2 -18164.519} C_VEL
LIN {X 0,Y 263.353,Z 249.144,A -85,B 0,C 180,E1 -18169.233,E2 -18169.233} C_VEL
LIN {X 0,Y 263.533,Z 249.132,A -85,B 0,C 180,E1 -18172.336,E2 -18172.336} C_VEL
LIN {X 0,Y 263.75,Z 249.101,A -85,B 0,C 180,E1 -18178.472,E2 -18178.472} C_VEL
LIN {X 0,Y 263.75,Z 249.095,A -85,B 0,C 180,E1 -18181.526,E2 -18181.526} C_VEL
LIN {X 0,Y 263.557,Z 249.135,A -85,B 0,C 180,E1 -18187.661,E2 -18187.661} C_VEL
LIN {X 0,Y 263.354,Z 249.141,A -85,B 0,C 180,E1 -18190.766,E2 -18190.766} C_VEL
LIN {X 0,Y 263.349,Z 249.179,A -85,B 0,C 180,E1 -18195.477,E2 -18195.477} C_VEL
LIN {X 0,Y 263.261,Z 249.161,A -85,B 0,C 180,E1 -18200.306,E2 -18200.306} C_VEL
LIN {X 0,Y 263.19,Z 249.189,A -85,B 0,C 180,E1 -18205.292,E2 -18205.292} C_VEL
LIN {X 0,Y 263.163,Z 249.182,A -85,B 0,C 180,E1 -18208.73,E2 -18208.73} C_VEL
LIN {X 0,Y 263.131,Z 249.203,A -85,B 0,C 180,E1 -18212.287,E2 -18212.287} C_VEL
LIN {X 0,Y 263.187,Z 249.188,A -85,B 0,C 180,E1 -18215.977,E2 -18215.977} C_VEL
LIN {X 0,Y 263.157,Z 249.189,A -85,B 0,C 180,E1 -18219.862,E2 -18219.862} C_VEL
LIN {X 0,Y 263.142,Z 249.204,A -85,B 0,C 180,E1 -18223.979,E2 -18223.979} C_VEL
LIN {X 0,Y 263.128,Z 249.15,A -85,B 0,C 180,E1 -18228.404,E2 -18228.404} C_VEL
LIN {X 0,Y 263.166,Z 249.206,A -85,B 0,C 180,E1 -18232.104,E2 -18232.104} C_VEL
LIN {X 0,Y 263.18,Z 249.165,A -85,B 0,C 180,E1 -18235.89,E2 -18235.89} C_VEL
LIN {X 0,Y 263.17,Z 249.409,A -85,B 0,C 180,E1 -18238.397,E2 -18238.397} C_VEL
LIN {X 0,Y 263.4,Z 250.377,A -85,B 0,C 180,E1 -18238.628,E2 -18238.628} C_VEL
LIN {X 0,Y 272.765,Z 267.863,A -85,B 0,C 180,E1 -18240.37,E2 -18240.37} C_VEL
LIN {X 0,Y 278.703,Z 278.173,A -85,B 0,C 180,E1 -18241.364,E2 -18241.364} C_VEL
LIN {X 0,Y 286.57,Z 289.242,A -85,B 0,C 180,E1 -18242.534,E2 -18242.534} C_VEL
LIN {X 0,Y 297.908,Z 301.87,A -85,B 0,C 180,E1 -18244.004,E2 -18244.004} C_VEL
LIN {X 0,Y 308.38,Z 312.099,A -85,B 0,C 180,E1 -18245.332,E2 -18245.332} C_VEL
LIN {X 0,Y 317.164,Z 320.091,A -85,B 0,C 180,E1 -18246.643,E2 -18246.643} C_VEL
LIN {X 0,Y 325.164,Z 327.151,A -85,B 0,C 180,E1 -18248.026,E2 -18248.026} C_VEL
LIN {X 0,Y 332.817,Z 333.59,A -85,B 0,C 180,E1 -18249.517,E2 -18249.517} C_VEL
LIN {X 0,Y 341.381,Z 340.247,A -85,B 0,C 180,E1 -18251.365,E2 -18251.365} C_VEL
LIN {X 0,Y 347.668,Z 345.167,A -85,B 0,C 180,E1 -18252.895,E2 -18252.895} C_VEL
LIN {X 0,Y 352.783,Z 348.849,A -85,B 0,C 180,E1 -18254.248,E2 -18254.248} C_VEL
LIN {X 0,Y 358.007,Z 352.867,A -85,B 0,C 180,E1 -18255.788,E2 -18255.788} C_VEL
LIN {X 0,Y 363.076,Z 356.031,A -85,B 0,C 180,E1 -18257.434,E2 -18257.434} C_VEL
LIN {X 0,Y 366.024,Z 357.794,A -85,B 0,C 180,E1 -18258.506,E2 -18258.506} C_VEL
LIN {X 0,Y 369.882,Z 360.941,A -85,B 0,C 180,E1 -18260.154,E2 -18260.154} C_VEL
LIN {X 0,Y 373.303,Z 363.219,A -85,B 0,C 180,E1 -18261.871,E2 -18261.871} C_VEL
LIN {X 0,Y 376.284,Z 364.842,A -85,B 0,C 180,E1 -18263.722,E2 -18263.722} C_VEL
LIN {X 0,Y 378.685,Z 365.813,A -85,B 0,C 180,E1 -18265.743,E2 -18265.743} C_VEL
LIN {X 0,Y 379.929,Z 366.268,A -85,B 0,C 180,E1 -18267.3,E2 -18267.3} C_VEL
LIN {X 0,Y 380.613,Z 366.688,A -85,B 0,C 180,E1 -18268.942,E2 -18268.942} C_VEL
LIN {X 0,Y 380.758,Z 366.623,A -85,B 0,C 180,E1 -18270,E2 -18270} C_VEL
LIN {X 0,Y 380.444,Z 366.566,A -85,B 0,C 180,E1 -18271.588,E2 -18271.588} C_VEL
LIN {X 0,Y 379.6,Z 366.062,A -85,B 0,C 180,E1 -18273.184,E2 -18273.184} C_VEL
LIN {X 0,Y 377.821,Z 365.521,A -85,B 0,C 180,E1 -18275.066,E2 -18275.066} C_VEL
LIN {X 0,Y 375.25,Z 364.306,A -85,B 0,C 180,E1 -18276.967,E2 -18276.967} C_VEL
LIN {X 0,Y 371.894,Z 362.31,A -85,B 0,C 180,E1 -18278.873,E2 -18278.873} C_VEL
LIN {X 0,Y 368.201,Z 359.657,A -85,B 0,C 180,E1 -18280.591,E2 -18280.591} C_VEL
LIN {X 0,Y 364.633,Z 356.872,A -85,B 0,C 180,E1 -18282.014,E2 -18282.014} C_VEL
LIN {X 0,Y 359.519,Z 353.857,A -85,B 0,C 180,E1 -18283.755,E2 -18283.755} C_VEL
LIN {X 0,Y 353.846,Z 349.699,A -85,B 0,C 180,E1 -18285.456,E2 -18285.456} C_VEL
LIN {X 0,Y 349.314,Z 346.263,A -85,B 0,C 180,E1 -18286.693,E2 -18286.693} C_VEL
LIN {X 0,Y 342.99,Z 341.645,A -85,B 0,C 180,E1 -18288.246,E2 -18288.246} C_VEL
LIN {X 0,Y 337.005,Z 336.832,A -85,B 0,C 180,E1 -18289.608,E2 -18289.608} C_VEL
LIN {X 0,Y 330.041,Z 331.141,A -85,B 0,C 180,E1 -18291.052,E2 -18291.052} C_VEL
LIN {X 0,Y 321.695,Z 324.119,A -85,B 0,C 180,E1 -18292.604,E2 -18292.604} C_VEL
LIN {X 0,Y 312.809,Z 316.139,A -85,B 0,C 180,E1 -18294.037,E2 -18294.037} C_VEL
LIN {X 0,Y 304.438,Z 308.298,A -85,B 0,C 180,E1 -18295.194,E2 -18295.194} C_VEL
LIN {X 0,Y 292.363,Z 295.966,A -85,B 0,C 180,E1 -18296.691,E2 -18296.691} C_VEL
LIN {X 0,Y 284.239,Z 286.146,A -85,B 0,C 180,E1 -18297.799,E2 -18297.799} C_VEL
LIN {X 0,Y 276.824,Z 275.282,A -85,B 0,C 180,E1 -18298.934,E2 -18298.934} C_VEL
LIN {X 0,Y 264.621,Z 252.753,A -85,B 0,C 180,E1 -18301.115,E2 -18301.115} C_VEL
LIN {X 0,Y 263.3,Z 250.051,A -85,B 0,C 180,E1 -18301.428,E2 -18301.428} C_VEL
LIN {X 0,Y 263.125,Z 249.264,A -85,B 0,C 180,E1 -18301.787,E2 -18301.787} C_VEL
LIN {X 0,Y 263.17,Z 249.166,A -85,B 0,C 180,E1 -18304.122,E2 -18304.122} C_VEL
LIN {X 0,Y 263.166,Z 249.206,A -85,B 0,C 180,E1 -18307.896,E2 -18307.896} C_VEL
LIN {X 0,Y 263.129,Z 249.149,A -85,B 0,C 180,E1 -18311.892,E2 -18311.892} C_VEL
LIN {X 0,Y 263.144,Z 249.205,A -85,B 0,C 180,E1 -18316.146,E2 -18316.146} C_VEL
LIN {X 0,Y 263.157,Z 249.189,A -85,B 0,C 180,E1 -18320.138,E2 -18320.138} C_VEL
LIN {X 0,Y 263.187,Z 249.188,A -85,B 0,C 180,E1 -18324.023,E2 -18324.023} C_VEL
LIN {X 0,Y 263.131,Z 249.203,A -85,B 0,C 180,E1 -18327.713,E2 -18327.713} C_VEL
LIN {X 0,Y 263.193,Z 249.172,A -85,B 0,C 180,E1 -18331.786,E2 -18331.786} C_VEL
LIN {X 0,Y 263.198,Z 249.193,A -85,B 0,C 180,E1 -18335.213,E2 -18335.213} C_VEL
LIN {X 0,Y 263.261,Z 249.161,A -85,B 0,C 180,E1 -18339.694,E2 -18339.694} C_VEL
LIN {X 0,Y 263.349,Z 249.179,A -85,B 0,C 180,E1 -18344.523,E2 -18344.523} C_VEL
LIN {X 0,Y 263.354,Z 249.141,A -85,B 0,C 180,E1 -18349.234,E2 -18349.234} C_VEL
LIN {X 0,Y 263.557,Z 249.135,A -85,B 0,C 180,E1 -18352.339,E2 -18352.339} C_VEL
LIN {X 0,Y 263.75,Z 249.095,A -85,B 0,C 180,E1 -18358.474,E2 -18358.474} C_VEL
LIN {X 0,Y 263.75,Z 249.101,A -85,B 0,C 180,E1 -18361.528,E2 -18361.528} C_VEL
LIN {X 0,Y 263.533,Z 249.132,A -85,B 0,C 180,E1 -18367.664,E2 -18367.664} C_VEL
LIN {X 0,Y 263.353,Z 249.144,A -85,B 0,C 180,E1 -18370.767,E2 -18370.767} C_VEL
LIN {X 0,Y 263.315,Z 249.177,A -85,B 0,C 180,E1 -18375.481,E2 -18375.481} C_VEL
LIN {X 0,Y 263.258,Z 249.167,A -85,B 0,C 180,E1 -18380.308,E2 -18380.308} C_VEL
LIN {X 0,Y 263.208,Z 249.179,A -85,B 0,C 180,E1 -18385.292,E2 -18385.292} C_VEL
LIN {X 0,Y 263.166,Z 249.188,A -85,B 0,C 180,E1 -18388.732,E2 -18388.732} C_VEL
LIN {X 0,Y 263.114,Z 249.193,A -85,B 0,C 180,E1 -18392.741,E2 -18392.741} C_VEL
LIN {X 0,Y 263.194,Z 249.2,A -85,B 0,C 180,E1 -18396.767,E2 -18396.767} C_VEL
LIN {X 0,Y 263.114,Z 249.196,A -85,B 0,C 180,E1 -18399.385,E2 -18399.385} C_VEL
LIN {X 0,Y 262.42,Z 249.283,A -85,B 0,C 180,E1 -18400.663,E2 -18400.663} C_VEL
LIN {X 0,Y 259.552,Z 249.654,A -85,B 0,C 180,E1 -18402.745,E2 -18402.745} C_VEL
LIN {X 0,Y 257.142,Z 249.95,A -85,B 0,C 180,E1 -18404.439,E2 -18404.439} C_VEL
LIN {X 0,Y 256.123,Z 250.078,A -85,B 0,C 180,E1 -18405.752,E2 -18405.752} C_VEL
LIN {X 0,Y 256.048,Z 250.088,A -85,B 0,C 180,E1 -18406.197,E2 -18406.197} C_VEL
LIN {X 0,Y 256.08,Z 250.081,A -85,B 0,C 180,E1 -18410.701,E2 -18410.701} C_VEL
LIN {X 0,Y 256.303,Z 250.931,A -85,B 0,C 180,E1 -18411.349,E2 -18411.349} C_VEL
LIN {X 0,Y 257.791,Z 257.618,A -85,B 0,C 180,E1 -18414.874,E2 -18414.874} C_VEL
LIN {X 0,Y 259.041,Z 263.926,A -85,B 0,C 180,E1 -18417.997,E2 -18417.997} C_VEL
LIN {X 0,Y 259.749,Z 266.081,A -85,B 0,C 180,E1 -18418.271,E2 -18418.271} C_VEL
LIN {X 0,Y 265.879,Z 279.837,A -85,B 0,C 180,E1 -18419.501,E2 -18419.501} C_VEL
LIN {X 0,Y 267.169,Z 284.086,A -85,B 0,C 180,E1 -18419.792,E2 -18419.792} C_VEL
LIN {X 0,Y 271.774,Z 308.003,A -85,B 0,C 180,E1 -18421.06,E2 -18421.06} C_VEL
LIN {X 0,Y 272.879,Z 315.466,A -85,B 0,C 180,E1 -18421.406,E2 -18421.406} C_VEL
LIN {X 0,Y 271.084,Z 370.562,A -85,B 0,C 180,E1 -18422.871,E2 -18422.871} C_VEL
LIN {X 0,Y 270.289,Z 380.719,A -85,B 0,C 180,E1 -18423.302,E2 -18423.302} C_VEL
LIN {X 0,Y 269.316,Z 390.169,A -85,B 0,C 180,E1 -18423.873,E2 -18423.873} C_VEL
LIN {X 0,Y 267.985,Z 400.248,A -85,B 0,C 180,E1 -18424.672,E2 -18424.672} C_VEL
LIN {X 0,Y 266.447,Z 410.003,A -85,B 0,C 180,E1 -18425.661,E2 -18425.661} C_VEL
LIN {X 0,Y 264.716,Z 420.069,A -85,B 0,C 180,E1 -18426.946,E2 -18426.946} C_VEL
LIN {X 0,Y 262.335,Z 431.564,A -85,B 0,C 180,E1 -18428.797,E2 -18428.797} C_VEL
LIN {X 0,Y 260.709,Z 439.401,A -85,B 0,C 180,E1 -18430.39,E2 -18430.39} C_VEL
LIN {X 0,Y 259.116,Z 446.993,A -85,B 0,C 180,E1 -18432.26,E2 -18432.26} C_VEL
LIN {X 0,Y 257.634,Z 453.442,A -85,B 0,C 180,E1 -18434.17,E2 -18434.17} C_VEL
LIN {X 0,Y 256.613,Z 457.943,A -85,B 0,C 180,E1 -18435.73,E2 -18435.73} C_VEL
LIN {X 0,Y 255.437,Z 463.436,A -85,B 0,C 180,E1 -18438.091,E2 -18438.091} C_VEL
LIN {X 0,Y 254.644,Z 467.764,A -85,B 0,C 180,E1 -18440.468,E2 -18440.468} C_VEL
LIN {X 0,Y 254.311,Z 470.133,A -85,B 0,C 180,E1 -18442.058,E2 -18442.058} C_VEL
LIN {X 0,Y 253.993,Z 473.119,A -85,B 0,C 180,E1 -18444.961,E2 -18444.961} C_VEL
LIN {X 0,Y 253.954,Z 474.387,A -85,B 0,C 180,E1 -18446.827,E2 -18446.827} C_VEL
LIN {X 0,Y 253.995,Z 474.979,A -85,B 0,C 180,E1 -18448.414,E2 -18448.414} C_VEL
LIN {X 0,Y 254.046,Z 475.136,A -85,B 0,C 180,E1 -18450,E2 -18450} C_VEL
LIN {X 0,Y 253.995,Z 474.979,A -85,B 0,C 180,E1 -18451.586,E2 -18451.586} C_VEL
LIN {X 0,Y 253.951,Z 474.387,A -85,B 0,C 180,E1 -18453.173,E2 -18453.173} C_VEL
LIN {X 0,Y 254.063,Z 471.934,A -85,B 0,C 180,E1 -18456.353,E2 -18456.353} C_VEL
LIN {X 0,Y 254.467,Z 468.982,A -85,B 0,C 180,E1 -18458.737,E2 -18458.737} C_VEL
LIN {X 0,Y 255.125,Z 464.99,A -85,B 0,C 180,E1 -18461.118,E2 -18461.118} C_VEL
LIN {X 0,Y 256.133,Z 459.858,A -85,B 0,C 180,E1 -18463.487,E2 -18463.487} C_VEL
LIN {X 0,Y 257.359,Z 454.598,A -85,B 0,C 180,E1 -18465.441,E2 -18465.441} C_VEL
LIN {X 0,Y 258.776,Z 448.281,A -85,B 0,C 180,E1 -18467.382,E2 -18467.382} C_VEL
LIN {X 0,Y 260.154,Z 442.001,A -85,B 0,C 180,E1 -18468.998,E2 -18468.998} C_VEL
LIN {X 0,Y 261.521,Z 435.402,A -85,B 0,C 180,E1 -18470.448,E2 -18470.448} C_VEL
LIN {X 0,Y 263.252,Z 427.225,A -85,B 0,C 180,E1 -18471.947,E2 -18471.947} C_VEL
LIN {X 0,Y 264.939,Z 418.717,A -85,B 0,C 180,E1 -18473.24,E2 -18473.24} C_VEL
LIN {X 0,Y 266.496,Z 410.004,A -85,B 0,C 180,E1 -18474.334,E2 -18474.334} C_VEL
LIN {X 0,Y 267.862,Z 401.255,A -85,B 0,C 180,E1 -18475.236,E2 -18475.236} C_VEL
LIN {X 0,Y 269.197,Z 391.457,A -85,B 0,C 180,E1 -18476.035,E2 -18476.035} C_VEL
LIN {X 0,Y 270.225,Z 381.564,A -85,B 0,C 180,E1 -18476.654,E2 -18476.654} C_VEL
LIN {X 0,Y 271.021,Z 371.792,A -85,B 0,C 180,E1 -18477.087,E2 -18477.087} C_VEL
LIN {X 0,Y 271.914,Z 347.649,A -85,B 0,C 180,E1 -18477.76,E2 -18477.76} C_VEL
LIN {X 0,Y 272.77,Z 314.277,A -85,B 0,C 180,E1 -18478.641,E2 -18478.641} C_VEL
LIN {X 0,Y 268.924,Z 292.518,A -85,B 0,C 180,E1 -18479.738,E2 -18479.738} C_VEL
LIN {X 0,Y 266.249,Z 280.787,A -85,B 0,C 180,E1 -18480.423,E2 -18480.423} C_VEL
LIN {X 0,Y 259.961,Z 266.487,A -85,B 0,C 180,E1 -18481.687,E2 -18481.687} C_VEL
LIN {X 0,Y 259.093,Z 264.116,A -85,B 0,C 180,E1 -18481.948,E2 -18481.948} C_VEL
LIN {X 0,Y 257.836,Z 258.03,A -85,B 0,C 180,E1 -18484.918,E2 -18484.918} C_VEL
LIN {X 0,Y 256.303,Z 250.933,A -85,B 0,C 180,E1 -18488.65,E2 -18488.65} C_VEL
LIN {X 0,Y 256.08,Z 250.08,A -85,B 0,C 180,E1 -18489.299,E2 -18489.299} C_VEL
LIN {X 0,Y 256.064,Z 250.089,A -85,B 0,C 180,E1 -18493.326,E2 -18493.326} C_VEL
LIN {X 0,Y 256.072,Z 250.088,A -85,B 0,C 180,E1 -18497.819,E2 -18497.819} C_VEL
LIN {X 0,Y 256.073,Z 250.074,A -85,B 0,C 180,E1 -18500.857,E2 -18500.857} C_VEL
LIN {X 0,Y 256.14,Z 250.08,A -85,B 0,C 180,E1 -18502.868,E2 -18502.868} C_VEL
LIN {X 0,Y 256.069,Z 250.065,A -85,B 0,C 180,E1 -18506.707,E2 -18506.707} C_VEL
LIN {X 0,Y 256.105,Z 250.08,A -85,B 0,C 180,E1 -18510.398,E2 -18510.398} C_VEL
LIN {X 0,Y 256.189,Z 250.055,A -85,B 0,C 180,E1 -18514.861,E2 -18514.861} C_VEL
LIN {X 0,Y 256.167,Z 250.057,A -85,B 0,C 180,E1 -18519.104,E2 -18519.104} C_VEL
LIN {X 0,Y 256.249,Z 250.053,A -85,B 0,C 180,E1 -18524.081,E2 -18524.081} C_VEL
LIN {X 0,Y 256.289,Z 250.049,A -85,B 0,C 180,E1 -18527.327,E2 -18527.327} C_VEL
LIN {X 0,Y 256.434,Z 249.998,A -85,B 0,C 180,E1 -18530.622,E2 -18530.622} C_VEL
LIN {X 0,Y 256.464,Z 250.031,A -85,B 0,C 180,E1 -18533.706,E2 -18533.706} C_VEL
LIN {X 0,Y 256.713,Z 249.978,A -85,B 0,C 180,E1 -18538.43,E2 -18538.43} C_VEL
LIN {X 0,Y 256.713,Z 249.971,A -85,B 0,C 180,E1 -18541.568,E2 -18541.568} C_VEL
LIN {X 0,Y 256.47,Z 250.026,A -85,B 0,C 180,E1 -18546.726,E2 -18546.726} C_VEL
LIN {X 0,Y 256.426,Z 250.001,A -85,B 0,C 180,E1 -18549.464,E2 -18549.464} C_VEL
LIN {X 0,Y 256.255,Z 250.064,A -85,B 0,C 180,E1 -18554.289,E2 -18554.289} C_VEL
LIN {X 0,Y 256.208,Z 250.044,A -85,B 0,C 180,E1 -18557.561,E2 -18557.561} C_VEL
LIN {X 0,Y 256.151,Z 250.057,A -85,B 0,C 180,E1 -18561.116,E2 -18561.116} C_VEL
LIN {X 0,Y 256.168,Z 250.065,A -85,B 0,C 180,E1 -18565.129,E2 -18565.129} C_VEL
LIN {X 0,Y 256.101,Z 250.076,A -85,B 0,C 180,E1 -18569.6,E2 -18569.6} C_VEL
LIN {X 0,Y 256.083,Z 250.069,A -85,B 0,C 180,E1 -18573.289,E2 -18573.289} C_VEL
LIN {X 0,Y 256.138,Z 250.08,A -85,B 0,C 180,E1 -18577.278,E2 -18577.278} C_VEL
LIN {X 0,Y 256.1,Z 250.065,A -85,B 0,C 180,E1 -18581.193,E2 -18581.193} C_VEL
LIN {X 0,Y 256.073,Z 250.079,A -85,B 0,C 180,E1 -18584.473,E2 -18584.473} C_VEL
LIN {X 0,Y 256.059,Z 250.032,A -85,B 0,C 180,E1 -18588.798,E2 -18588.798} C_VEL
LIN {X 0,Y 256.145,Z 250.069,A -85,B 0,C 180,E1 -18592.87,E2 -18592.87} C_VEL
LIN {X 0,Y 256.097,Z 250.11,A -85,B 0,C 180,E1 -18597.302,E2 -18597.302} C_VEL
LIN {X 0,Y 256.254,Z 250.963,A -85,B 0,C 180,E1 -18597.642,E2 -18597.642} C_VEL
LIN {X 0,Y 257.769,Z 253.868,A -85,B 0,C 180,E1 -18597.99,E2 -18597.99} C_VEL
LIN {X 0,Y 266.043,Z 269.057,A -85,B 0,C 180,E1 -18599.573,E2 -18599.573} C_VEL
LIN {X 0,Y 272.725,Z 281.291,A -85,B 0,C 180,E1 -18600.763,E2 -18600.763} C_VEL
LIN {X 0,Y 281.448,Z 293.701,A -85,B 0,C 180,E1 -18602.112,E2 -18602.112} C_VEL
LIN {X 0,Y 291.044,Z 304.558,A -85,B 0,C 180,E1 -18603.41,E2 -18603.41} C_VEL
LIN {X 0,Y 303.455,Z 316.955,A -85,B 0,C 180,E1 -18604.939,E2 -18604.939} C_VEL
LIN {X 0,Y 312.641,Z 325.188,A -85,B 0,C 180,E1 -18606.195,E2 -18606.195} C_VEL
LIN {X 0,Y 321.75,Z 333.036,A -85,B 0,C 180,E1 -18607.663,E2 -18607.663} C_VEL
LIN {X 0,Y 330.541,Z 340.273,A -85,B 0,C 180,E1 -18609.312,E2 -18609.312} C_VEL
LIN {X 0,Y 339.212,Z 346.92,A -85,B 0,C 180,E1 -18611.146,E2 -18611.146} C_VEL
LIN {X 0,Y 345.908,Z 352.019,A -85,B 0,C 180,E1 -18612.729,E2 -18612.729} C_VEL
LIN {X 0,Y 350.538,Z 355.276,A -85,B 0,C 180,E1 -18613.919,E2 -18613.919} C_VEL
LIN {X 0,Y 355.955,Z 359.405,A -85,B 0,C 180,E1 -18615.477,E2 -18615.477} C_VEL
LIN {X 0,Y 360.956,Z 362.534,A -85,B 0,C 180,E1 -18617.039,E2 -18617.039} C_VEL
LIN {X 0,Y 364.571,Z 364.711,A -85,B 0,C 180,E1 -18618.329,E2 -18618.329} C_VEL
LIN {X 0,Y 368.887,Z 368.055,A -85,B 0,C 180,E1 -18620.127,E2 -18620.127} C_VEL
LIN {X 0,Y 372.365,Z 370.282,A -85,B 0,C 180,E1 -18621.851,E2 -18621.851} C_VEL
LIN {X 0,Y 375.376,Z 371.893,A -85,B 0,C 180,E1 -18623.707,E2 -18623.707} C_VEL
LIN {X 0,Y 377.255,Z 372.685,A -85,B 0,C 180,E1 -18625.198,E2 -18625.198} C_VEL
LIN {X 0,Y 379.058,Z 373.315,A -85,B 0,C 180,E1 -18627.294,E2 -18627.294} C_VEL
LIN {X 0,Y 379.744,Z 373.734,A -85,B 0,C 180,E1 -18628.94,E2 -18628.94} C_VEL
LIN {X 0,Y 379.893,Z 373.67,A -85,B 0,C 180,E1 -18630,E2 -18630} C_VEL
LIN {X 0,Y 379.625,Z 373.632,A -85,B 0,C 180,E1 -18631.43,E2 -18631.43} C_VEL
LIN {X 0,Y 378.724,Z 373.102,A -85,B 0,C 180,E1 -18633.191,E2 -18633.191} C_VEL
LIN {X 0,Y 376.928,Z 372.568,A -85,B 0,C 180,E1 -18635.078,E2 -18635.078} C_VEL
LIN {X 0,Y 374.242,Z 371.319,A -85,B 0,C 180,E1 -18637.04,E2 -18637.04} C_VEL
LIN {X 0,Y 370.772,Z 369.318,A -85,B 0,C 180,E1 -18638.978,E2 -18638.978} C_VEL
LIN {X 0,Y 366.9,Z 366.587,A -85,B 0,C 180,E1 -18640.737,E2 -18640.737} C_VEL
LIN {X 0,Y 363.238,Z 363.737,A -85,B 0,C 180,E1 -18642.174,E2 -18642.174} C_VEL
LIN {X 0,Y 358.36,Z 360.954,A -85,B 0,C 180,E1 -18643.8,E2 -18643.8} C_VEL
LIN {X 0,Y 352.641,Z 356.98,A -85,B 0,C 180,E1 -18645.489,E2 -18645.489} C_VEL
LIN {X 0,Y 347.918,Z 353.356,A -85,B 0,C 180,E1 -18646.763,E2 -18646.763} C_VEL
LIN {X 0,Y 341.393,Z 348.733,A -85,B 0,C 180,E1 -18648.349,E2 -18648.349} C_VEL
LIN {X 0,Y 335.048,Z 343.707,A -85,B 0,C 180,E1 -18649.763,E2 -18649.763} C_VEL
LIN {X 0,Y 327.939,Z 338.085,A -85,B 0,C 180,E1 -18651.204,E2 -18651.204} C_VEL
LIN {X 0,Y 319.005,Z 330.738,A -85,B 0,C 180,E1 -18652.799,E2 -18652.799} C_VEL
LIN {X 0,Y 311.301,Z 323.983,A -85,B 0,C 180,E1 -18654,E2 -18654} C_VEL
LIN {X 0,Y 302.067,Z 315.669,A -85,B 0,C 180,E1 -18655.238,E2 -18655.238} C_VEL
LIN {X 0,Y 287.707,Z 301.057,A -85,B 0,C 180,E1 -18657.022,E2 -18657.022} C_VEL
LIN {X 0,Y 279.434,Z 291.038,A -85,B 0,C 180,E1 -18658.184,E2 -18658.184} C_VEL
LIN {X 0,Y 271.559,Z 279.405,A -85,B 0,C 180,E1 -18659.432,E2 -18659.432} C_VEL
LIN {X 0,Y 259.58,Z 257.092,A -85,B 0,C 180,E1 -18661.656,E2 -18661.656} C_VEL
LIN {X 0,Y 256.314,Z 251.129,A -85,B 0,C 180,E1 -18662.335,E2 -18662.335} C_VEL
LIN {X 0,Y 256.098,Z 250.151,A -85,B 0,C 180,E1 -18662.699,E2 -18662.699} C_VEL
LIN {X 0,Y 256.118,Z 250.044,A -85,B 0,C 180,E1 -18665.187,E2 -18665.187} C_VEL
LIN {X 0,Y 256.086,Z 250.066,A -85,B 0,C 180,E1 -18669.139,E2 -18669.139} C_VEL
LIN {X 0,Y 256.07,Z 250.035,A -85,B 0,C 180,E1 -18673.325,E2 -18673.325} C_VEL
LIN {X 0,Y 256.122,Z 250.072,A -85,B 0,C 180,E1 -18677.806,E2 -18677.806} C_VEL
LIN {X 0,Y 256.106,Z 250.075,A -85,B 0,C 180,E1 -18680.865,E2 -18680.865} C_VEL
LIN {X 0,Y 256.119,Z 250.06,A -85,B 0,C 180,E1 -18684.814,E2 -18684.814} C_VEL
LIN {X 0,Y 256.09,Z 250.086,A -85,B 0,C 180,E1 -18688.573,E2 -18688.573} C_VEL
LIN {X 0,Y 256.135,Z 250.048,A -85,B 0,C 180,E1 -18692.196,E2 -18692.196} C_VEL
LIN {X 0,Y 256.14,Z 250.076,A -85,B 0,C 180,E1 -18695.697,E2 -18695.697} C_VEL
LIN {X 0,Y 256.16,Z 250.053,A -85,B 0,C 180,E1 -18699.105,E2 -18699.105} C_VEL
LIN {X 0,Y 256.299,Z 250.055,A -85,B 0,C 180,E1 -18704.086,E2 -18704.086} C_VEL
LIN {X 0,Y 256.294,Z 250.046,A -85,B 0,C 180,E1 -18707.329,E2 -18707.329} C_VEL
LIN {X 0,Y 256.514,Z 250.008,A -85,B 0,C 180,E1 -18712.127,E2 -18712.127} C_VEL
LIN {X 0,Y 256.498,Z 250.021,A -85,B 0,C 180,E1 -18716.86,E2 -18716.86} C_VEL
LIN {X 0,Y 256.757,Z 249.957,A -85,B 0,C 180,E1 -18720.001,E2 -18720.001} C_VEL
LIN {X 0,Y 256.495,Z 250.027,A -85,B 0,C 180,E1 -18723.142,E2 -18723.142} C_VEL
LIN {X 0,Y 256.474,Z 250.007,A -85,B 0,C 180,E1 -18727.876,E2 -18727.876} C_VEL
LIN {X 0,Y 256.295,Z 250.026,A -85,B 0,C 180,E1 -18731.067,E2 -18731.067} C_VEL
LIN {X 0,Y 256.236,Z 250.064,A -85,B 0,C 180,E1 -18734.292,E2 -18734.292} C_VEL
LIN {X 0,Y 256.182,Z 250.039,A -85,B 0,C 180,E1 -18737.565,E2 -18737.565} C_VEL
LIN {X 0,Y 256.158,Z 250.061,A -85,B 0,C 180,E1 -18741.12,E2 -18741.12} C_VEL
LIN {X 0,Y 256.189,Z 250.055,A -85,B 0,C 180,E1 -18745.139,E2 -18745.139} C_VEL
LIN {X 0,Y 256.105,Z 250.08,A -85,B 0,C 180,E1 -18749.602,E2 -18749.602} C_VEL
LIN {X 0,Y 256.069,Z 250.065,A -85,B 0,C 180,E1 -18753.293,E2 -18753.293} C_VEL
LIN {X 0,Y 256.124,Z 250.081,A -85,B 0,C 180,E1 -18757.274,E2 -18757.274} C_VEL
LIN {X 0,Y 256.056,Z 250.08,A -85,B 0,C 180,E1 -18761.204,E2 -18761.204} C_VEL
LIN {X 0,Y 256.056,Z 250.084,A -85,B 0,C 180,E1 -18765.532,E2 -18765.532} C_VEL
LIN {X 0,Y 256.048,Z 250.088,A -85,B 0,C 180,E1 -18766.197,E2 -18766.197} C_VEL
LIN {X 0,Y 255.346,Z 250.186,A -85,B 0,C 180,E1 -18767.089,E2 -18767.089} C_VEL
LIN {X 0,Y 252.41,Z 250.515,A -85,B 0,C 180,E1 -18768.49,E2 -18768.49} C_VEL
LIN {X 0,Y 249.684,Z 251.028,A -85,B 0,C 180,E1 -18769.89,E2 -18769.89} C_VEL
LIN {X 0,Y 249.238,Z 251.82,A -85,B 0,C 180,E1 -18770.614,E2 -18770.614} C_VEL
LIN {X 0,Y 249.277,Z 252.051,A -85,B 0,C 180,E1 -18770.755,E2 -18770.755} C_VEL
LIN {X 0,Y 250.604,Z 257.801,A -85,B 0,C 180,E1 -18773.919,E2 -18773.919} C_VEL
LIN {X 0,Y 251.82,Z 263.755,A -85,B 0,C 180,E1 -18776.98,E2 -18776.98} C_VEL
LIN {X 0,Y 253.179,Z 267.139,A -85,B 0,C 180,E1 -18777.389,E2 -18777.389} C_VEL
LIN {X 0,Y 260.086,Z 282.638,A -85,B 0,C 180,E1 -18778.841,E2 -18778.841} C_VEL
LIN {X 0,Y 261.328,Z 286.784,A -85,B 0,C 180,E1 -18779.134,E2 -18779.134} C_VEL
LIN {X 0,Y 265.741,Z 310.327,A -85,B 0,C 180,E1 -18780.415,E2 -18780.415} C_VEL
LIN {X 0,Y 266.618,Z 316.546,A -85,B 0,C 180,E1 -18780.709,E2 -18780.709} C_VEL
LIN {X 0,Y 264.84,Z 369.713,A -85,B 0,C 180,E1 -18782.148,E2 -18782.148} C_VEL
LIN {X 0,Y 264.057,Z 379.864,A -85,B 0,C 180,E1 -18782.58,E2 -18782.58} C_VEL
LIN {X 0,Y 262.966,Z 389.976,A -85,B 0,C 180,E1 -18783.192,E2 -18783.192} C_VEL
LIN {X 0,Y 261.574,Z 400.055,A -85,B 0,C 180,E1 -18784.006,E2 -18784.006} C_VEL
LIN {X 0,Y 260,Z 409.81,A -85,B 0,C 180,E1 -18785.017,E2 -18785.017} C_VEL
LIN {X 0,Y 258.179,Z 419.876,A -85,B 0,C 180,E1 -18786.327,E2 -18786.327} C_VEL
LIN {X 0,Y 255.734,Z 431.371,A -85,B 0,C 180,E1 -18788.223,E2 -18788.223} C_VEL
LIN {X 0,Y 253.707,Z 440.509,A -85,B 0,C 180,E1 -18790.163,E2 -18790.163} C_VEL
LIN {X 0,Y 252.011,Z 448.088,A -85,B 0,C 180,E1 -18792.136,E2 -18792.136} C_VEL
LIN {X 0,Y 250.505,Z 454.404,A -85,B 0,C 180,E1 -18794.125,E2 -18794.125} C_VEL
LIN {X 0,Y 249.202,Z 459.664,A -85,B 0,C 180,E1 -18796.13,E2 -18796.13} C_VEL
LIN {X 0,Y 248.136,Z 464.797,A -85,B 0,C 180,E1 -18798.565,E2 -18798.565} C_VEL
LIN {X 0,Y 247.412,Z 468.788,A -85,B 0,C 180,E1 -18801.012,E2 -18801.012} C_VEL
LIN {X 0,Y 247.011,Z 471.742,A -85,B 0,C 180,E1 -18803.465,E2 -18803.465} C_VEL
LIN {X 0,Y 246.858,Z 474.194,A -85,B 0,C 180,E1 -18806.736,E2 -18806.736} C_VEL
LIN {X 0,Y 246.905,Z 474.787,A -85,B 0,C 180,E1 -18808.369,E2 -18808.369} C_VEL
LIN {X 0,Y 246.976,Z 474.944,A -85,B 0,C 180,E1 -18810,E2 -18810} C_VEL
LIN {X 0,Y 246.904,Z 474.787,A -85,B 0,C 180,E1 -18811.631,E2 -18811.631} C_VEL
LIN {X 0,Y 246.855,Z 474.194,A -85,B 0,C 180,E1 -18813.264,E2 -18813.264} C_VEL
LIN {X 0,Y 246.985,Z 471.741,A -85,B 0,C 180,E1 -18816.536,E2 -18816.536} C_VEL
LIN {X 0,Y 247.412,Z 468.788,A -85,B 0,C 180,E1 -18818.988,E2 -18818.988} C_VEL
LIN {X 0,Y 248.136,Z 464.797,A -85,B 0,C 180,E1 -18821.435,E2 -18821.435} C_VEL
LIN {X 0,Y 249.202,Z 459.664,A -85,B 0,C 180,E1 -18823.87,E2 -18823.87} C_VEL
LIN {X 0,Y 250.5,Z 454.404,A -85,B 0,C 180,E1 -18825.875,E2 -18825.875} C_VEL
LIN {X 0,Y 252.007,Z 448.088,A -85,B 0,C 180,E1 -18827.865,E2 -18827.865} C_VEL
LIN {X 0,Y 253.709,Z 440.509,A -85,B 0,C 180,E1 -18829.836,E2 -18829.836} C_VEL
LIN {X 0,Y 255.714,Z 431.371,A -85,B 0,C 180,E1 -18831.779,E2 -18831.779} C_VEL
LIN {X 0,Y 258.181,Z 419.876,A -85,B 0,C 180,E1 -18833.673,E2 -18833.673} C_VEL
LIN {X 0,Y 260.011,Z 409.811,A -85,B 0,C 180,E1 -18834.982,E2 -18834.982} C_VEL
LIN {X 0,Y 261.578,Z 400.055,A -85,B 0,C 180,E1 -18835.994,E2 -18835.994} C_VEL
LIN {X 0,Y 262.991,Z 389.977,A -85,B 0,C 180,E1 -18836.805,E2 -18836.805} C_VEL
LIN {X 0,Y 264.068,Z 379.855,A -85,B 0,C 180,E1 -18837.42,E2 -18837.42} C_VEL
LIN {X 0,Y 264.835,Z 369.629,A -85,B 0,C 180,E1 -18837.854,E2 -18837.854} C_VEL
LIN {X 0,Y 266.545,Z 315.386,A -85,B 0,C 180,E1 -18839.335,E2 -18839.335} C_VEL
LIN {X 0,Y 262.629,Z 293.052,A -85,B 0,C 180,E1 -18840.503,E2 -18840.503} C_VEL
LIN {X 0,Y 260.391,Z 283.44,A -85,B 0,C 180,E1 -18841.094,E2 -18841.094} C_VEL
LIN {X 0,Y 253.184,Z 267.147,A -85,B 0,C 180,E1 -18842.61,E2 -18842.61} C_VEL
LIN {X 0,Y 251.819,Z 263.749,A -85,B 0,C 180,E1 -18843.019,E2 -18843.019} C_VEL
LIN {X 0,Y 250.206,Z 256.021,A -85,B 0,C 180,E1 -18847.05,E2 -18847.05} C_VEL
LIN {X 0,Y 249.024,Z 250.991,A -85,B 0,C 180,E1 -18849.945,E2 -18849.945} C_VEL
LIN {X 0,Y 249.011,Z 250.958,A -85,B 0,C 180,E1 -18852.792,E2 -18852.792} C_VEL
LIN {X 0,Y 249.011,Z 250.968,A -85,B 0,C 180,E1 -18857.361,E2 -18857.361} C_VEL
LIN {X 0,Y 249.03,Z 250.958,A -85,B 0,C 180,E1 -18861.619,E2 -18861.619} C_VEL
LIN {X 0,Y 249.047,Z 250.937,A -85,B 0,C 180,E1 -18865.639,E2 -18865.639} C_VEL
LIN {X 0,Y 249.049,Z 250.964,A -85,B 0,C 180,E1 -18869.472,E2 -18869.472} C_VEL
LIN {X 0,Y 249.072,Z 250.926,A -85,B 0,C 180,E1 -18873.161,E2 -18873.161} C_VEL
LIN {X 0,Y 249.08,Z 250.956,A -85,B 0,C 180,E1 -18876.732,E2 -18876.732} C_VEL
LIN {X 0,Y 249.1,Z 250.921,A -85,B 0,C 180,E1 -18880.21,E2 -18880.21} C_VEL
LIN {X 0,Y 249.196,Z 250.923,A -85,B 0,C 180,E1 -18883.618,E2 -18883.618} C_VEL
LIN {X 0,Y 249.242,Z 250.908,A -85,B 0,C 180,E1 -18888.615,E2 -18888.615} C_VEL
LIN {X 0,Y 249.422,Z 250.88,A -85,B 0,C 180,E1 -18891.9,E2 -18891.9} C_VEL
LIN {X 0,Y 249.288,Z 250.934,A -85,B 0,C 180,E1 -18895.147,E2 -18895.147} C_VEL
LIN {X 0,Y 249.675,Z 250.854,A -85,B 0,C 180,E1 -18898.386,E2 -18898.386} C_VEL
LIN {X 0,Y 249.675,Z 250.847,A -85,B 0,C 180,E1 -18901.612,E2 -18901.612} C_VEL
LIN {X 0,Y 249.44,Z 250.902,A -85,B 0,C 180,E1 -18906.71,E2 -18906.71} C_VEL
LIN {X 0,Y 249.342,Z 250.882,A -85,B 0,C 180,E1 -18909.736,E2 -18909.736} C_VEL
LIN {X 0,Y 249.205,Z 250.944,A -85,B 0,C 180,E1 -18914.702,E2 -18914.702} C_VEL
LIN {X 0,Y 249.136,Z 250.917,A -85,B 0,C 180,E1 -18918.077,E2 -18918.077} C_VEL
LIN {X 0,Y 249.082,Z 250.944,A -85,B 0,C 180,E1 -18921.518,E2 -18921.518} C_VEL
LIN {X 0,Y 249.114,Z 250.937,A -85,B 0,C 180,E1 -18925.474,E2 -18925.474} C_VEL
LIN {X 0,Y 249.071,Z 250.939,A -85,B 0,C 180,E1 -18928.988,E2 -18928.988} C_VEL
LIN {X 0,Y 249.034,Z 250.958,A -85,B 0,C 180,E1 -18932.424,E2 -18932.424} C_VEL
LIN {X 0,Y 249.073,Z 250.949,A -85,B 0,C 180,E1 -18936.337,E2 -18936.337} C_VEL
LIN {X 0,Y 249.075,Z 250.939,A -85,B 0,C 180,E1 -18940.463,E2 -18940.463} C_VEL
LIN {X 0,Y 249.016,Z 250.948,A -85,B 0,C 180,E1 -18944.875,E2 -18944.875} C_VEL
LIN {X 0,Y 249.022,Z 250.905,A -85,B 0,C 180,E1 -18947.364,E2 -18947.364} C_VEL
LIN {X 0,Y 249.037,Z 250.963,A -85,B 0,C 180,E1 -18951.622,E2 -18951.622} C_VEL
LIN {X 0,Y 249.058,Z 250.921,A -85,B 0,C 180,E1 -18955.642,E2 -18955.642} C_VEL
LIN {X 0,Y 249.09,Z 251.186,A -85,B 0,C 180,E1 -18956.447,E2 -18956.447} C_VEL
LIN {X 0,Y 249.432,Z 252.507,A -85,B 0,C 180,E1 -18956.718,E2 -18956.718} C_VEL
LIN {X 0,Y 258.639,Z 268.948,A -85,B 0,C 180,E1 -18958.594,E2 -18958.594} C_VEL
LIN {X 0,Y 267.083,Z 284.798,A -85,B 0,C 180,E1 -18960.185,E2 -18960.185} C_VEL
LIN {X 0,Y 275.387,Z 296.916,A -85,B 0,C 180,E1 -18961.531,E2 -18961.531} C_VEL
LIN {X 0,Y 285.68,Z 308.961,A -85,B 0,C 180,E1 -18962.988,E2 -18962.988} C_VEL
LIN {X 0,Y 299.415,Z 322.62,A -85,B 0,C 180,E1 -18964.69,E2 -18964.69} C_VEL
LIN {X 0,Y 308.98,Z 331.091,A -85,B 0,C 180,E1 -18965.924,E2 -18965.924} C_VEL
LIN {X 0,Y 316.306,Z 337.307,A -85,B 0,C 180,E1 -18967.018,E2 -18967.018} C_VEL
LIN {X 0,Y 322.882,Z 342.524,A -85,B 0,C 180,E1 -18968.12,E2 -18968.12} C_VEL
LIN {X 0,Y 329.769,Z 348.123,A -85,B 0,C 180,E1 -18969.414,E2 -18969.414} C_VEL
LIN {X 0,Y 336.917,Z 353.532,A -85,B 0,C 180,E1 -18970.902,E2 -18970.902} C_VEL
LIN {X 0,Y 344.054,Z 358.803,A -85,B 0,C 180,E1 -18972.543,E2 -18972.543} C_VEL
LIN {X 0,Y 349.787,Z 362.918,A -85,B 0,C 180,E1 -18974.013,E2 -18974.013} C_VEL
LIN {X 0,Y 355.469,Z 366.991,A -85,B 0,C 180,E1 -18975.643,E2 -18975.643} C_VEL
LIN {X 0,Y 360.385,Z 369.879,A -85,B 0,C 180,E1 -18977.176,E2 -18977.176} C_VEL
LIN {X 0,Y 363.495,Z 371.875,A -85,B 0,C 180,E1 -18978.292,E2 -18978.292} C_VEL
LIN {X 0,Y 367.635,Z 374.985,A -85,B 0,C 180,E1 -18980.004,E2 -18980.004} C_VEL
LIN {X 0,Y 371.055,Z 377.162,A -85,B 0,C 180,E1 -18981.674,E2 -18981.674} C_VEL
LIN {X 0,Y 374.16,Z 378.811,A -85,B 0,C 180,E1 -18983.529,E2 -18983.529} C_VEL
LIN {X 0,Y 376.273,Z 379.716,A -85,B 0,C 180,E1 -18985.185,E2 -18985.185} C_VEL
LIN {X 0,Y 377.957,Z 380.268,A -85,B 0,C 180,E1 -18987.069,E2 -18987.069} C_VEL
LIN {X 0,Y 378.778,Z 380.767,A -85,B 0,C 180,E1 -18988.937,E2 -18988.937} C_VEL
LIN {X 0,Y 378.931,Z 380.692,A -85,B 0,C 180,E1 -18990,E2 -18990} C_VEL
LIN {X 0,Y 378.672,Z 380.667,A -85,B 0,C 180,E1 -18991.434,E2 -18991.434} C_VEL
LIN {X 0,Y 377.772,Z 380.12,A -85,B 0,C 180,E1 -18993.199,E2 -18993.199} C_VEL
LIN {X 0,Y 375.953,Z 379.603,A -85,B 0,C 180,E1 -18995.091,E2 -18995.091} C_VEL
LIN {X 0,Y 373.246,Z 378.363,A -85,B 0,C 180,E1 -18997.059,E2 -18997.059} C_VEL
LIN {X 0,Y 369.921,Z 376.473,A -85,B 0,C 180,E1 -18998.916,E2 -18998.916} C_VEL
LIN {X 0,Y 365.986,Z 373.828,A -85,B 0,C 180,E1 -19000.715,E2 -19000.715} C_VEL
LIN {X 0,Y 361.438,Z 370.457,A -85,B 0,C 180,E1 -19002.458,E2 -19002.458} C_VEL
LIN {X 0,Y 356.567,Z 367.679,A -85,B 0,C 180,E1 -19004.027,E2 -19004.027} C_VEL
LIN {X 0,Y 351.157,Z 363.984,A -85,B 0,C 180,E1 -19005.602,E2 -19005.602} C_VEL
LIN {X 0,Y 344.956,Z 359.4,A -85,B 0,C 180,E1 -19007.233,E2 -19007.233} C_VEL
LIN {X 0,Y 337.822,Z 354.294,A -85,B 0,C 180,E1 -19008.895,E2 -19008.895} C_VEL
LIN {X 0,Y 331.658,Z 349.541,A -85,B 0,C 180,E1 -19010.205,E2 -19010.205} C_VEL
LIN {X 0,Y 324.959,Z 344.306,A -85,B 0,C 180,E1 -19011.493,E2 -19011.493} C_VEL
LIN {X 0,Y 317.715,Z 338.528,A -85,B 0,C 180,E1 -19012.753,E2 -19012.753} C_VEL
LIN {X 0,Y 309.729,Z 331.684,A -85,B 0,C 180,E1 -19013.972,E2 -19013.972} C_VEL
LIN {X 0,Y 301.357,Z 324.318,A -85,B 0,C 180,E1 -19015.078,E2 -19015.078} C_VEL
LIN {X 0,Y 288.844,Z 312.325,A -85,B 0,C 180,E1 -19016.598,E2 -19016.598} C_VEL
LIN {X 0,Y 276.865,Z 298.86,A -85,B 0,C 180,E1 -19018.246,E2 -19018.246} C_VEL
LIN {X 0,Y 267.701,Z 285.801,A -85,B 0,C 180,E1 -19019.708,E2 -19019.708} C_VEL
LIN {X 0,Y 260.785,Z 273.116,A -85,B 0,C 180,E1 -19020.985,E2 -19020.985} C_VEL
LIN {X 0,Y 254.284,Z 261.065,A -85,B 0,C 180,E1 -19022.27,E2 -19022.27} C_VEL
LIN {X 0,Y 250.463,Z 254.396,A -85,B 0,C 180,E1 -19023.051,E2 -19023.051} C_VEL
LIN {X 0,Y 249.202,Z 251.705,A -85,B 0,C 180,E1 -19023.399,E2 -19023.399} C_VEL
LIN {X 0,Y 249.044,Z 250.988,A -85,B 0,C 180,E1 -19023.777,E2 -19023.777} C_VEL
LIN {X 0,Y 249.055,Z 250.964,A -85,B 0,C 180,E1 -19027.805,E2 -19027.805} C_VEL
LIN {X 0,Y 249.024,Z 250.915,A -85,B 0,C 180,E1 -19030.474,E2 -19030.474} C_VEL
LIN {X 0,Y 249.016,Z 250.942,A -85,B 0,C 180,E1 -19034.876,E2 -19034.876} C_VEL
LIN {X 0,Y 249.059,Z 250.957,A -85,B 0,C 180,E1 -19037.373,E2 -19037.373} C_VEL
LIN {X 0,Y 249.05,Z 250.962,A -85,B 0,C 180,E1 -19041.625,E2 -19041.625} C_VEL
LIN {X 0,Y 249.059,Z 250.936,A -85,B 0,C 180,E1 -19045.643,E2 -19045.643} C_VEL
LIN {X 0,Y 249.045,Z 250.963,A -85,B 0,C 180,E1 -19049.473,E2 -19049.473} C_VEL
LIN {X 0,Y 249.065,Z 250.928,A -85,B 0,C 180,E1 -19053.162,E2 -19053.162} C_VEL
LIN {X 0,Y 249.059,Z 250.961,A -85,B 0,C 180,E1 -19056.732,E2 -19056.732} C_VEL
LIN {X 0,Y 249.105,Z 250.918,A -85,B 0,C 180,E1 -19060.212,E2 -19060.212} C_VEL
LIN {X 0,Y 249.241,Z 250.928,A -85,B 0,C 180,E1 -19063.623,E2 -19063.623} C_VEL
LIN {X 0,Y 249.244,Z 250.904,A -85,B 0,C 180,E1 -19068.617,E2 -19068.617} C_VEL
LIN {X 0,Y 249.454,Z 250.883,A -85,B 0,C 180,E1 -19071.903,E2 -19071.903} C_VEL
LIN {X 0,Y 249.296,Z 250.933,A -85,B 0,C 180,E1 -19075.149,E2 -19075.149} C_VEL
LIN {X 0,Y 249.675,Z 250.847,A -85,B 0,C 180,E1 -19078.388,E2 -19078.388} C_VEL
LIN {X 0,Y 249.675,Z 250.854,A -85,B 0,C 180,E1 -19081.614,E2 -19081.614} C_VEL
LIN {X 0,Y 249.434,Z 250.903,A -85,B 0,C 180,E1 -19086.472,E2 -19086.472} C_VEL
LIN {X 0,Y 249.343,Z 250.88,A -85,B 0,C 180,E1 -19089.737,E2 -19089.737} C_VEL
LIN {X 0,Y 249.179,Z 250.943,A -85,B 0,C 180,E1 -19094.706,E2 -19094.706} C_VEL
LIN {X 0,Y 249.118,Z 250.914,A -85,B 0,C 180,E1 -19098.08,E2 -19098.08} C_VEL
LIN {X 0,Y 249.088,Z 250.947,A -85,B 0,C 180,E1 -19101.519,E2 -19101.519} C_VEL
LIN {X 0,Y 249.131,Z 250.928,A -85,B 0,C 180,E1 -19105.482,E2 -19105.482} C_VEL
LIN {X 0,Y 249.074,Z 250.945,A -85,B 0,C 180,E1 -19108.99,E2 -19108.99} C_VEL
LIN {X 0,Y 249.032,Z 250.951,A -85,B 0,C 180,E1 -19112.427,E2 -19112.427} C_VEL
LIN {X 0,Y 249.056,Z 250.956,A -85,B 0,C 180,E1 -19116.342,E2 -19116.342} C_VEL
LIN {X 0,Y 249.008,Z 250.951,A -85,B 0,C 180,E1 -19120.479,E2 -19120.479} C_VEL
LIN {X 0,Y 248.995,Z 250.958,A -85,B 0,C 180,E1 -19124.882,E2 -19124.882} C_VEL
LIN {X 0,Y 249.018,Z 250.955,A -85,B 0,C 180,E1 -19127.364,E2 -19127.364} C_VEL
LIN {X 0,Y 249.042,Z 251.095,A -85,B 0,C 180,E1 -19130.19,E2 -19130.19} C_VEL
LIN {X 0,Y 249.277,Z 252.051,A -85,B 0,C 180,E1 -19130.755,E2 -19130.755} C_VEL
LIN {X 0,Y 249.001,Z 253.725,A -85,B 0,C 180,E1 -19131.578,E2 -19131.578} C_VEL
LIN {X 0,Y 246.795,Z 256.877,A -85,B 0,C 180,E1 -19132.853,E2 -19132.853} C_VEL
LIN {X 0,Y 244.517,Z 260.039,A -85,B 0,C 180,E1 -19134.151,E2 -19134.151} C_VEL
LIN {X 0,Y 244.164,Z 261.749,A -85,B 0,C 180,E1 -19134.996,E2 -19134.996} C_VEL
LIN {X 0,Y 244.603,Z 263.712,A -85,B 0,C 180,E1 -19135.917,E2 -19135.917} C_VEL
LIN {X 0,Y 246.384,Z 267.66,A -85,B 0,C 180,E1 -19136.398,E2 -19136.398} C_VEL
LIN {X 0,Y 253.872,Z 284.471,A -85,B 0,C 180,E1 -19138.055,E2 -19138.055} C_VEL
LIN {X 0,Y 255.363,Z 288.742,A -85,B 0,C 180,E1 -19138.4,E2 -19138.4} C_VEL
LIN {X 0,Y 259.611,Z 311.566,A -85,B 0,C 180,E1 -19139.688,E2 -19139.688} C_VEL
LIN {X 0,Y 260.363,Z 316.459,A -85,B 0,C 180,E1 -19139.937,E2 -19139.937} C_VEL
LIN {X 0,Y 258.563,Z 370.104,A -85,B 0,C 180,E1 -19141.436,E2 -19141.436} C_VEL
LIN {X 0,Y 257.681,Z 380.698,A -85,B 0,C 180,E1 -19141.907,E2 -19141.907} C_VEL
LIN {X 0,Y 256.507,Z 391.072,A -85,B 0,C 180,E1 -19142.572,E2 -19142.572} C_VEL
LIN {X 0,Y 254.748,Z 402.882,A -85,B 0,C 180,E1 -19143.586,E2 -19143.586} C_VEL
LIN {X 0,Y 252.749,Z 414.278,A -85,B 0,C 180,E1 -19144.91,E2 -19144.91} C_VEL
LIN {X 0,Y 250.654,Z 424.572,A -85,B 0,C 180,E1 -19146.45,E2 -19146.45} C_VEL
LIN {X 0,Y 248.655,Z 433.096,A -85,B 0,C 180,E1 -19148.007,E2 -19148.007} C_VEL
LIN {X 0,Y 246.993,Z 440.315,A -85,B 0,C 180,E1 -19149.601,E2 -19149.601} C_VEL
LIN {X 0,Y 245.667,Z 446.253,A -85,B 0,C 180,E1 -19151.142,E2 -19151.142} C_VEL
LIN {X 0,Y 243.923,Z 453.055,A -85,B 0,C 180,E1 -19153.254,E2 -19153.254} C_VEL
LIN {X 0,Y 242.807,Z 457.556,A -85,B 0,C 180,E1 -19154.9,E2 -19154.9} C_VEL
LIN {X 0,Y 241.468,Z 463.048,A -85,B 0,C 180,E1 -19157.391,E2 -19157.391} C_VEL
LIN {X 0,Y 240.605,Z 467.377,A -85,B 0,C 180,E1 -19159.906,E2 -19159.906} C_VEL
LIN {X 0,Y 240.21,Z 469.747,A -85,B 0,C 180,E1 -19161.588,E2 -19161.588} C_VEL
LIN {X 0,Y 239.928,Z 471.548,A -85,B 0,C 180,E1 -19163.271,E2 -19163.271} C_VEL
LIN {X 0,Y 239.764,Z 474.001,A -85,B 0,C 180,E1 -19166.639,E2 -19166.639} C_VEL
LIN {X 0,Y 239.816,Z 474.594,A -85,B 0,C 180,E1 -19168.321,E2 -19168.321} C_VEL
LIN {X 0,Y 239.884,Z 474.751,A -85,B 0,C 180,E1 -19170,E2 -19170} C_VEL
LIN {X 0,Y 239.816,Z 474.594,A -85,B 0,C 180,E1 -19171.679,E2 -19171.679} C_VEL
LIN {X 0,Y 239.762,Z 474.001,A -85,B 0,C 180,E1 -19173.361,E2 -19173.361} C_VEL
LIN {X 0,Y 239.908,Z 471.548,A -85,B 0,C 180,E1 -19176.729,E2 -19176.729} C_VEL
LIN {X 0,Y 240.378,Z 468.595,A -85,B 0,C 180,E1 -19179.254,E2 -19179.254} C_VEL
LIN {X 0,Y 241.157,Z 464.603,A -85,B 0,C 180,E1 -19181.771,E2 -19181.771} C_VEL
LIN {X 0,Y 242.287,Z 459.471,A -85,B 0,C 180,E1 -19184.274,E2 -19184.274} C_VEL
LIN {X 0,Y 243.652,Z 454.211,A -85,B 0,C 180,E1 -19186.334,E2 -19186.334} C_VEL
LIN {X 0,Y 245.234,Z 447.895,A -85,B 0,C 180,E1 -19188.375,E2 -19188.375} C_VEL
LIN {X 0,Y 246.638,Z 441.943,A -85,B 0,C 180,E1 -19189.995,E2 -19189.995} C_VEL
LIN {X 0,Y 248.203,Z 435.014,A -85,B 0,C 180,E1 -19191.599,E2 -19191.599} C_VEL
LIN {X 0,Y 250.106,Z 426.839,A -85,B 0,C 180,E1 -19193.166,E2 -19193.166} C_VEL
LIN {X 0,Y 251.935,Z 418.331,A -85,B 0,C 180,E1 -19194.516,E2 -19194.516} C_VEL
LIN {X 0,Y 253.583,Z 409.618,A -85,B 0,C 180,E1 -19195.661,E2 -19195.661} C_VEL
LIN {X 0,Y 255.213,Z 399.862,A -85,B 0,C 180,E1 -19196.693,E2 -19196.693} C_VEL
LIN {X 0,Y 256.535,Z 391.072,A -85,B 0,C 180,E1 -19197.425,E2 -19197.425} C_VEL
LIN {X 0,Y 257.686,Z 380.703,A -85,B 0,C 180,E1 -19198.093,E2 -19198.093} C_VEL
LIN {X 0,Y 258.468,Z 371.347,A -85,B 0,C 180,E1 -19198.523,E2 -19198.523} C_VEL
LIN {X 0,Y 259.534,Z 344.719,A -85,B 0,C 180,E1 -19199.288,E2 -19199.288} C_VEL
LIN {X 0,Y 260.36,Z 316.518,A -85,B 0,C 180,E1 -19200.062,E2 -19200.062} C_VEL
LIN {X 0,Y 256.633,Z 294.982,A -85,B 0,C 180,E1 -19201.227,E2 -19201.227} C_VEL
LIN {X 0,Y 254.697,Z 286.41,A -85,B 0,C 180,E1 -19201.767,E2 -19201.767} C_VEL
LIN {X 0,Y 247.876,Z 270.915,A -85,B 0,C 180,E1 -19203.265,E2 -19203.265} C_VEL
LIN {X 0,Y 244.647,Z 263.971,A -85,B 0,C 180,E1 -19204.036,E2 -19204.036} C_VEL
LIN {X 0,Y 244.338,Z 262.67,A -85,B 0,C 180,E1 -19204.507,E2 -19204.507} C_VEL
LIN {X 0,Y 242.825,Z 255.355,A -85,B 0,C 180,E1 -19208.605,E2 -19208.605} C_VEL
LIN {X 0,Y 241.978,Z 251.916,A -85,B 0,C 180,E1 -19210.671,E2 -19210.671} C_VEL
LIN {X 0,Y 241.928,Z 251.845,A -85,B 0,C 180,E1 -19214.202,E2 -19214.202} C_VEL
LIN {X 0,Y 241.936,Z 251.847,A -85,B 0,C 180,E1 -19218.076,E2 -19218.076} C_VEL
LIN {X 0,Y 241.996,Z 251.841,A -85,B 0,C 180,E1 -19222.418,E2 -19222.418} C_VEL
LIN {X 0,Y 241.983,Z 251.817,A -85,B 0,C 180,E1 -19226.507,E2 -19226.507} C_VEL
LIN {X 0,Y 242.015,Z 251.83,A -85,B 0,C 180,E1 -19230.596,E2 -19230.596} C_VEL
LIN {X 0,Y 242.069,Z 251.803,A -85,B 0,C 180,E1 -19234.182,E2 -19234.182} C_VEL
LIN {X 0,Y 242.054,Z 251.825,A -85,B 0,C 180,E1 -19238.296,E2 -19238.296} C_VEL
LIN {X 0,Y 242.116,Z 251.801,A -85,B 0,C 180,E1 -19243.315,E2 -19243.315} C_VEL
LIN {X 0,Y 242.154,Z 251.817,A -85,B 0,C 180,E1 -19246.573,E2 -19246.573} C_VEL
LIN {X 0,Y 242.343,Z 251.751,A -85,B 0,C 180,E1 -19250.403,E2 -19250.403} C_VEL
LIN {X 0,Y 242.404,Z 251.776,A -85,B 0,C 180,E1 -19253.339,E2 -19253.339} C_VEL
LIN {X 0,Y 242.635,Z 251.731,A -85,B 0,C 180,E1 -19258.339,E2 -19258.339} C_VEL
LIN {X 0,Y 242.636,Z 251.724,A -85,B 0,C 180,E1 -19261.659,E2 -19261.659} C_VEL
LIN {X 0,Y 242.421,Z 251.779,A -85,B 0,C 180,E1 -19266.682,E2 -19266.682} C_VEL
LIN {X 0,Y 242.267,Z 251.762,A -85,B 0,C 180,E1 -19270.023,E2 -19270.023} C_VEL
LIN {X 0,Y 242.166,Z 251.818,A -85,B 0,C 180,E1 -19275.14,E2 -19275.14} C_VEL
LIN {X 0,Y 242.07,Z 251.793,A -85,B 0,C 180,E1 -19278.623,E2 -19278.623} C_VEL
LIN {X 0,Y 242.005,Z 251.833,A -85,B 0,C 180,E1 -19282.18,E2 -19282.18} C_VEL
LIN {X 0,Y 242.065,Z 251.808,A -85,B 0,C 180,E1 -19285.837,E2 -19285.837} C_VEL
LIN {X 0,Y 242.005,Z 251.829,A -85,B 0,C 180,E1 -19289.582,E2 -19289.582} C_VEL
LIN {X 0,Y 241.989,Z 251.821,A -85,B 0,C 180,E1 -19293.49,E2 -19293.49} C_VEL
LIN {X 0,Y 242.011,Z 251.841,A -85,B 0,C 180,E1 -19297.577,E2 -19297.577} C_VEL
LIN {X 0,Y 241.982,Z 251.829,A -85,B 0,C 180,E1 -19301.912,E2 -19301.912} C_VEL
LIN {X 0,Y 241.94,Z 251.806,A -85,B 0,C 180,E1 -19305.8,E2 -19305.8} C_VEL
LIN {X 0,Y 241.971,Z 251.806,A -85,B 0,C 180,E1 -19310.284,E2 -19310.284} C_VEL
LIN {X 0,Y 242.033,Z 251.799,A -85,B 0,C 180,E1 -19314.497,E2 -19314.497} C_VEL
LIN {X 0,Y 242.076,Z 252.075,A -85,B 0,C 180,E1 -19315.364,E2 -19315.364} C_VEL
LIN {X 0,Y 242.428,Z 253.434,A -85,B 0,C 180,E1 -19315.65,E2 -19315.65} C_VEL
LIN {X 0,Y 251.851,Z 269.917,A -85,B 0,C 180,E1 -19317.671,E2 -19317.671} C_VEL
LIN {X 0,Y 261.767,Z 288.773,A -85,B 0,C 180,E1 -19319.635,E2 -19319.635} C_VEL
LIN {X 0,Y 269.723,Z 300.577,A -85,B 0,C 180,E1 -19320.981,E2 -19320.981} C_VEL
LIN {X 0,Y 279.098,Z 312.005,A -85,B 0,C 180,E1 -19322.378,E2 -19322.378} C_VEL
LIN {X 0,Y 293.795,Z 326.898,A -85,B 0,C 180,E1 -19324.277,E2 -19324.277} C_VEL
LIN {X 0,Y 305.831,Z 337.429,A -85,B 0,C 180,E1 -19325.732,E2 -19325.732} C_VEL
LIN {X 0,Y 314.872,Z 344.964,A -85,B 0,C 180,E1 -19327.04,E2 -19327.04} C_VEL
LIN {X 0,Y 322.413,Z 350.915,A -85,B 0,C 180,E1 -19328.288,E2 -19328.288} C_VEL
LIN {X 0,Y 329.771,Z 356.471,A -85,B 0,C 180,E1 -19329.669,E2 -19329.669} C_VEL
LIN {X 0,Y 338.338,Z 362.976,A -85,B 0,C 180,E1 -19331.489,E2 -19331.489} C_VEL
LIN {X 0,Y 346.117,Z 368.283,A -85,B 0,C 180,E1 -19333.348,E2 -19333.348} C_VEL
LIN {X 0,Y 352.036,Z 372.654,A -85,B 0,C 180,E1 -19334.958,E2 -19334.958} C_VEL
LIN {X 0,Y 357.688,Z 376.167,A -85,B 0,C 180,E1 -19336.686,E2 -19336.686} C_VEL
LIN {X 0,Y 361.257,Z 378.272,A -85,B 0,C 180,E1 -19337.912,E2 -19337.912} C_VEL
LIN {X 0,Y 365.803,Z 381.719,A -85,B 0,C 180,E1 -19339.774,E2 -19339.774} C_VEL
LIN {X 0,Y 369.47,Z 384.031,A -85,B 0,C 180,E1 -19341.541,E2 -19341.541} C_VEL
LIN {X 0,Y 372.788,Z 385.762,A -85,B 0,C 180,E1 -19343.505,E2 -19343.505} C_VEL
LIN {X 0,Y 374.924,Z 386.669,A -85,B 0,C 180,E1 -19345.168,E2 -19345.168} C_VEL
LIN {X 0,Y 376.632,Z 387.228,A -85,B 0,C 180,E1 -19347.059,E2 -19347.059} C_VEL
LIN {X 0,Y 377.443,Z 387.74,A -85,B 0,C 180,E1 -19348.933,E2 -19348.933} C_VEL
LIN {X 0,Y 377.607,Z 387.667,A -85,B 0,C 180,E1 -19350,E2 -19350} C_VEL
LIN {X 0,Y 377.311,Z 387.606,A -85,B 0,C 180,E1 -19351.601,E2 -19351.601} C_VEL
LIN {X 0,Y 376.473,Z 387.096,A -85,B 0,C 180,E1 -19353.21,E2 -19353.21} C_VEL
LIN {X 0,Y 374.605,Z 386.556,A -85,B 0,C 180,E1 -19355.109,E2 -19355.109} C_VEL
LIN {X 0,Y 371.872,Z 385.318,A -85,B 0,C 180,E1 -19357.085,E2 -19357.085} C_VEL
LIN {X 0,Y 368.483,Z 383.459,A -85,B 0,C 180,E1 -19358.951,E2 -19358.951} C_VEL
LIN {X 0,Y 364.543,Z 380.868,A -85,B 0,C 180,E1 -19360.758,E2 -19360.758} C_VEL
LIN {X 0,Y 359.989,Z 377.387,A -85,B 0,C 180,E1 -19362.544,E2 -19362.544} C_VEL
LIN {X 0,Y 354.468,Z 374.229,A -85,B 0,C 180,E1 -19364.32,E2 -19364.32} C_VEL
LIN {X 0,Y 348.255,Z 369.958,A -85,B 0,C 180,E1 -19366.089,E2 -19366.089} C_VEL
LIN {X 0,Y 342.477,Z 365.764,A -85,B 0,C 180,E1 -19367.556,E2 -19367.556} C_VEL
LIN {X 0,Y 335.202,Z 360.644,A -85,B 0,C 180,E1 -19369.2,E2 -19369.2} C_VEL
LIN {X 0,Y 328.999,Z 355.907,A -85,B 0,C 180,E1 -19370.484,E2 -19370.484} C_VEL
LIN {X 0,Y 322.054,Z 350.621,A -85,B 0,C 180,E1 -19371.776,E2 -19371.776} C_VEL
LIN {X 0,Y 313.108,Z 343.554,A -85,B 0,C 180,E1 -19373.239,E2 -19373.239} C_VEL
LIN {X 0,Y 303.511,Z 335.458,A -85,B 0,C 180,E1 -19374.562,E2 -19374.562} C_VEL
LIN {X 0,Y 291.165,Z 324.365,A -85,B 0,C 180,E1 -19376.043,E2 -19376.043} C_VEL
LIN {X 0,Y 278.281,Z 311.068,A -85,B 0,C 180,E1 -19377.738,E2 -19377.738} C_VEL
LIN {X 0,Y 269.723,Z 300.588,A -85,B 0,C 180,E1 -19379.019,E2 -19379.019} C_VEL
LIN {X 0,Y 261.389,Z 288.161,A -85,B 0,C 180,E1 -19380.433,E2 -19380.433} C_VEL
LIN {X 0,Y 249.381,Z 265.515,A -85,B 0,C 180,E1 -19382.839,E2 -19382.839} C_VEL
LIN {X 0,Y 243.428,Z 255.269,A -85,B 0,C 180,E1 -19384.113,E2 -19384.113} C_VEL
LIN {X 0,Y 242.164,Z 252.525,A -85,B 0,C 180,E1 -19384.492,E2 -19384.492} C_VEL
LIN {X 0,Y 242.026,Z 251.847,A -85,B 0,C 180,E1 -19384.936,E2 -19384.936} C_VEL
LIN {X 0,Y 242.005,Z 251.838,A -85,B 0,C 180,E1 -19388.364,E2 -19388.364} C_VEL
LIN {X 0,Y 241.946,Z 251.784,A -85,B 0,C 180,E1 -19391.92,E2 -19391.92} C_VEL
LIN {X 0,Y 241.989,Z 251.843,A -85,B 0,C 180,E1 -19396.557,E2 -19396.557} C_VEL
LIN {X 0,Y 242.005,Z 251.823,A -85,B 0,C 180,E1 -19400.292,E2 -19400.292} C_VEL
LIN {X 0,Y 242.034,Z 251.815,A -85,B 0,C 180,E1 -19404.498,E2 -19404.498} C_VEL
LIN {X 0,Y 241.973,Z 251.845,A -85,B 0,C 180,E1 -19408.481,E2 -19408.481} C_VEL
LIN {X 0,Y 241.998,Z 251.807,A -85,B 0,C 180,E1 -19412.313,E2 -19412.313} C_VEL
LIN {X 0,Y 242.039,Z 251.835,A -85,B 0,C 180,E1 -19416.015,E2 -19416.015} C_VEL
LIN {X 0,Y 242.033,Z 251.804,A -85,B 0,C 180,E1 -19419.609,E2 -19419.609} C_VEL
LIN {X 0,Y 242.162,Z 251.806,A -85,B 0,C 180,E1 -19423.279,E2 -19423.279} C_VEL
LIN {X 0,Y 242.18,Z 251.787,A -85,B 0,C 180,E1 -19428.28,E2 -19428.28} C_VEL
LIN {X 0,Y 242.4,Z 251.757,A -85,B 0,C 180,E1 -19431.666,E2 -19431.666} C_VEL
LIN {X 0,Y 242.257,Z 251.809,A -85,B 0,C 180,E1 -19435.008,E2 -19435.008} C_VEL
LIN {X 0,Y 242.636,Z 251.724,A -85,B 0,C 180,E1 -19438.341,E2 -19438.341} C_VEL
LIN {X 0,Y 242.635,Z 251.731,A -85,B 0,C 180,E1 -19441.661,E2 -19441.661} C_VEL
LIN {X 0,Y 242.404,Z 251.776,A -85,B 0,C 180,E1 -19446.661,E2 -19446.661} C_VEL
LIN {X 0,Y 242.267,Z 251.762,A -85,B 0,C 180,E1 -19450.025,E2 -19450.025} C_VEL
LIN {X 0,Y 242.137,Z 251.816,A -85,B 0,C 180,E1 -19455.144,E2 -19455.144} C_VEL
LIN {X 0,Y 242.058,Z 251.791,A -85,B 0,C 180,E1 -19458.626,E2 -19458.626} C_VEL
LIN {X 0,Y 242.014,Z 251.834,A -85,B 0,C 180,E1 -19462.181,E2 -19462.181} C_VEL
LIN {X 0,Y 242.068,Z 251.803,A -85,B 0,C 180,E1 -19465.839,E2 -19465.839} C_VEL
LIN {X 0,Y 242.008,Z 251.834,A -85,B 0,C 180,E1 -19469.584,E2 -19469.584} C_VEL
LIN {X 0,Y 241.983,Z 251.817,A -85,B 0,C 180,E1 -19473.493,E2 -19473.493} C_VEL
LIN {X 0,Y 241.996,Z 251.841,A -85,B 0,C 180,E1 -19477.582,E2 -19477.582} C_VEL
LIN {X 0,Y 241.936,Z 251.847,A -85,B 0,C 180,E1 -19481.924,E2 -19481.924} C_VEL
LIN {X 0,Y 241.935,Z 251.851,A -85,B 0,C 180,E1 -19486.572,E2 -19486.572} C_VEL
LIN {X 0,Y 242.007,Z 252.008,A -85,B 0,C 180,E1 -19489.422,E2 -19489.422} C_VEL
LIN {X 0,Y 243.63,Z 258.842,A -85,B 0,C 180,E1 -19493.385,E2 -19493.385} C_VEL
LIN {X 0,Y 244.164,Z 261.749,A -85,B 0,C 180,E1 -19494.996,E2 -19494.996} C_VEL
LIN {X 0,Y 244.735,Z 263.895,A -85,B 0,C 180,E1 -19495.696,E2 -19495.696} C_VEL
LIN {X 0,Y 245.624,Z 266.899,A -85,B 0,C 180,E1 -19496.191,E2 -19496.191} C_VEL
LIN {X 0,Y 247.039,Z 272.288,A -85,B 0,C 180,E1 -19496.656,E2 -19496.656} C_VEL
LIN {X 0,Y 248.997,Z 288.803,A -85,B 0,C 180,E1 -19497.502,E2 -19497.502} C_VEL
LIN {X 0,Y 249.462,Z 290.811,A -85,B 0,C 180,E1 -19497.637,E2 -19497.637} C_VEL
LIN {X 0,Y 253.502,Z 312.901,A -85,B 0,C 180,E1 -19498.927,E2 -19498.927} C_VEL
LIN {X 0,Y 254.228,Z 318.911,A -85,B 0,C 180,E1 -19499.218,E2 -19499.218} C_VEL
LIN {X 0,Y 252.39,Z 369.371,A -85,B 0,C 180,E1 -19500.645,E2 -19500.645} C_VEL
LIN {X 0,Y 251.529,Z 379.892,A -85,B 0,C 180,E1 -19501.116,E2 -19501.116} C_VEL
LIN {X 0,Y 250.37,Z 389.591,A -85,B 0,C 180,E1 -19501.726,E2 -19501.726} C_VEL
LIN {X 0,Y 248.905,Z 399.67,A -85,B 0,C 180,E1 -19502.575,E2 -19502.575} C_VEL
LIN {X 0,Y 247.51,Z 407.794,A -85,B 0,C 180,E1 -19503.435,E2 -19503.435} C_VEL
LIN {X 0,Y 245.761,Z 416.787,A -85,B 0,C 180,E1 -19504.599,E2 -19504.599} C_VEL
LIN {X 0,Y 243.867,Z 425.512,A -85,B 0,C 180,E1 -19505.979,E2 -19505.979} C_VEL
LIN {X 0,Y 242.076,Z 432.903,A -85,B 0,C 180,E1 -19507.376,E2 -19507.376} C_VEL
LIN {X 0,Y 240.307,Z 440.121,A -85,B 0,C 180,E1 -19509.007,E2 -19509.007} C_VEL
LIN {X 0,Y 238.844,Z 446.355,A -85,B 0,C 180,E1 -19510.678,E2 -19510.678} C_VEL
LIN {X 0,Y 237.083,Z 452.86,A -85,B 0,C 180,E1 -19512.756,E2 -19512.756} C_VEL
LIN {X 0,Y 235.929,Z 457.362,A -85,B 0,C 180,E1 -19514.449,E2 -19514.449} C_VEL
LIN {X 0,Y 234.512,Z 462.854,A -85,B 0,C 180,E1 -19517.011,E2 -19517.011} C_VEL
LIN {X 0,Y 233.579,Z 467.183,A -85,B 0,C 180,E1 -19519.599,E2 -19519.599} C_VEL
LIN {X 0,Y 233.177,Z 469.554,A -85,B 0,C 180,E1 -19521.332,E2 -19521.332} C_VEL
LIN {X 0,Y 232.874,Z 471.355,A -85,B 0,C 180,E1 -19523.067,E2 -19523.067} C_VEL
LIN {X 0,Y 232.674,Z 473.809,A -85,B 0,C 180,E1 -19526.537,E2 -19526.537} C_VEL
LIN {X 0,Y 232.729,Z 474.402,A -85,B 0,C 180,E1 -19528.27,E2 -19528.27} C_VEL
LIN {X 0,Y 232.795,Z 474.559,A -85,B 0,C 180,E1 -19530,E2 -19530} C_VEL
LIN {X 0,Y 232.729,Z 474.402,A -85,B 0,C 180,E1 -19531.73,E2 -19531.73} C_VEL
LIN {X 0,Y 232.689,Z 473.13,A -85,B 0,C 180,E1 -19534.637,E2 -19534.637} C_VEL
LIN {X 0,Y 232.831,Z 471.354,A -85,B 0,C 180,E1 -19536.935,E2 -19536.935} C_VEL
LIN {X 0,Y 233.363,Z 468.402,A -85,B 0,C 180,E1 -19539.534,E2 -19539.534} C_VEL
LIN {X 0,Y 234.17,Z 464.41,A -85,B 0,C 180,E1 -19542.127,E2 -19542.127} C_VEL
LIN {X 0,Y 235.39,Z 459.278,A -85,B 0,C 180,E1 -19544.701,E2 -19544.701} C_VEL
LIN {X 0,Y 236.817,Z 454.017,A -85,B 0,C 180,E1 -19546.819,E2 -19546.819} C_VEL
LIN {X 0,Y 238.477,Z 447.701,A -85,B 0,C 180,E1 -19548.915,E2 -19548.915} C_VEL
LIN {X 0,Y 239.94,Z 441.749,A -85,B 0,C 180,E1 -19550.578,E2 -19550.578} C_VEL
LIN {X 0,Y 241.604,Z 434.821,A -85,B 0,C 180,E1 -19552.219,E2 -19552.219} C_VEL
LIN {X 0,Y 243.588,Z 426.646,A -85,B 0,C 180,E1 -19553.824,E2 -19553.824} C_VEL
LIN {X 0,Y 245.496,Z 418.138,A -85,B 0,C 180,E1 -19555.204,E2 -19555.204} C_VEL
LIN {X 0,Y 247.188,Z 409.424,A -85,B 0,C 180,E1 -19556.375,E2 -19556.375} C_VEL
LIN {X 0,Y 248.906,Z 399.67,A -85,B 0,C 180,E1 -19557.425,E2 -19557.425} C_VEL
LIN {X 0,Y 250.247,Z 390.879,A -85,B 0,C 180,E1 -19558.175,E2 -19558.175} C_VEL
LIN {X 0,Y 251.442,Z 380.711,A -85,B 0,C 180,E1 -19558.842,E2 -19558.842} C_VEL
LIN {X 0,Y 252.307,Z 370.574,A -85,B 0,C 180,E1 -19559.311,E2 -19559.311} C_VEL
LIN {X 0,Y 253.491,Z 340.776,A -85,B 0,C 180,E1 -19560.177,E2 -19560.177} C_VEL
LIN {X 0,Y 254.145,Z 317.078,A -85,B 0,C 180,E1 -19560.852,E2 -19560.852} C_VEL
LIN {X 0,Y 250.399,Z 295.54,A -85,B 0,C 180,E1 -19562.071,E2 -19562.071} C_VEL
LIN {X 0,Y 249.004,Z 289.281,A -85,B 0,C 180,E1 -19562.48,E2 -19562.48} C_VEL
LIN {X 0,Y 242.23,Z 273.943,A -85,B 0,C 180,E1 -19564.033,E2 -19564.033} C_VEL
LIN {X 0,Y 238.722,Z 266.757,A -85,B 0,C 180,E1 -19564.856,E2 -19564.856} C_VEL
LIN {X 0,Y 237.291,Z 263.414,A -85,B 0,C 180,E1 -19565.298,E2 -19565.298} C_VEL
LIN {X 0,Y 236.451,Z 259.25,A -85,B 0,C 180,E1 -19567.565,E2 -19567.565} C_VEL
LIN {X 0,Y 234.912,Z 252.747,A -85,B 0,C 180,E1 -19571.586,E2 -19571.586} C_VEL
LIN {X 0,Y 234.89,Z 252.714,A -85,B 0,C 180,E1 -19575.897,E2 -19575.897} C_VEL
LIN {X 0,Y 234.883,Z 252.715,A -85,B 0,C 180,E1 -19578.831,E2 -19578.831} C_VEL
LIN {X 0,Y 234.922,Z 252.709,A -85,B 0,C 180,E1 -19581.078,E2 -19581.078} C_VEL
LIN {X 0,Y 234.935,Z 252.694,A -85,B 0,C 180,E1 -19585.362,E2 -19585.362} C_VEL
LIN {X 0,Y 234.924,Z 252.723,A -85,B 0,C 180,E1 -19589.43,E2 -19589.43} C_VEL
LIN {X 0,Y 234.995,Z 252.68,A -85,B 0,C 180,E1 -19593.793,E2 -19593.793} C_VEL
LIN {X 0,Y 235.01,Z 252.693,A -85,B 0,C 180,E1 -19598.969,E2 -19598.969} C_VEL
LIN {X 0,Y 235.057,Z 252.675,A -85,B 0,C 180,E1 -19603.091,E2 -19603.091} C_VEL
LIN {X 0,Y 235.11,Z 252.677,A -85,B 0,C 180,E1 -19607.921,E2 -19607.921} C_VEL
LIN {X 0,Y 235.314,Z 252.63,A -85,B 0,C 180,E1 -19611.411,E2 -19611.411} C_VEL
LIN {X 0,Y 235.209,Z 252.686,A -85,B 0,C 180,E1 -19614.856,E2 -19614.856} C_VEL
LIN {X 0,Y 235.595,Z 252.607,A -85,B 0,C 180,E1 -19618.29,E2 -19618.29} C_VEL
LIN {X 0,Y 235.595,Z 252.6,A -85,B 0,C 180,E1 -19621.708,E2 -19621.708} C_VEL
LIN {X 0,Y 235.392,Z 252.653,A -85,B 0,C 180,E1 -19626.858,E2 -19626.858} C_VEL
LIN {X 0,Y 235.214,Z 252.64,A -85,B 0,C 180,E1 -19630.327,E2 -19630.327} C_VEL
LIN {X 0,Y 235.113,Z 252.697,A -85,B 0,C 180,E1 -19635.605,E2 -19635.605} C_VEL
LIN {X 0,Y 235.005,Z 252.671,A -85,B 0,C 180,E1 -19639.205,E2 -19639.205} C_VEL
LIN {X 0,Y 234.951,Z 252.719,A -85,B 0,C 180,E1 -19642.883,E2 -19642.883} C_VEL
LIN {X 0,Y 234.965,Z 252.684,A -85,B 0,C 180,E1 -19646.657,E2 -19646.657} C_VEL
LIN {X 0,Y 234.921,Z 252.723,A -85,B 0,C 180,E1 -19650.568,E2 -19650.568} C_VEL
LIN {X 0,Y 234.958,Z 252.692,A -85,B 0,C 180,E1 -19654.632,E2 -19654.632} C_VEL
LIN {X 0,Y 234.964,Z 252.709,A -85,B 0,C 180,E1 -19658.951,E2 -19658.951} C_VEL
LIN {X 0,Y 234.962,Z 252.719,A -85,B 0,C 180,E1 -19663.467,E2 -19663.467} C_VEL
LIN {X 0,Y 234.893,Z 252.662,A -85,B 0,C 180,E1 -19668.416,E2 -19668.416} C_VEL
LIN {X 0,Y 234.952,Z 252.697,A -85,B 0,C 180,E1 -19671.085,E2 -19671.085} C_VEL
LIN {X 0,Y 235.007,Z 252.927,A -85,B 0,C 180,E1 -19674.156,E2 -19674.156} C_VEL
LIN {X 0,Y 235.261,Z 253.899,A -85,B 0,C 180,E1 -19674.444,E2 -19674.444} C_VEL
LIN {X 0,Y 236.743,Z 256.566,A -85,B 0,C 180,E1 -19674.823,E2 -19674.823} C_VEL
LIN {X 0,Y 246.481,Z 273.554,A -85,B 0,C 180,E1 -19676.996,E2 -19676.996} C_VEL
LIN {X 0,Y 256.533,Z 292.853,A -85,B 0,C 180,E1 -19679.073,E2 -19679.073} C_VEL
LIN {X 0,Y 264.555,Z 304.857,A -85,B 0,C 180,E1 -19680.484,E2 -19680.484} C_VEL
LIN {X 0,Y 273.021,Z 315.426,A -85,B 0,C 180,E1 -19681.803,E2 -19681.803} C_VEL
LIN {X 0,Y 285.041,Z 328.005,A -85,B 0,C 180,E1 -19683.449,E2 -19683.449} C_VEL
LIN {X 0,Y 294.128,Z 336.435,A -85,B 0,C 180,E1 -19684.561,E2 -19684.561} C_VEL
LIN {X 0,Y 303.26,Z 344.248,A -85,B 0,C 180,E1 -19685.65,E2 -19685.65} C_VEL
LIN {X 0,Y 313.036,Z 352.229,A -85,B 0,C 180,E1 -19686.996,E2 -19686.996} C_VEL
LIN {X 0,Y 321.108,Z 358.525,A -85,B 0,C 180,E1 -19688.331,E2 -19688.331} C_VEL
LIN {X 0,Y 329.091,Z 364.26,A -85,B 0,C 180,E1 -19689.837,E2 -19689.837} C_VEL
LIN {X 0,Y 336.245,Z 369.795,A -85,B 0,C 180,E1 -19691.374,E2 -19691.374} C_VEL
LIN {X 0,Y 343.931,Z 375.037,A -85,B 0,C 180,E1 -19693.204,E2 -19693.204} C_VEL
LIN {X 0,Y 350.387,Z 379.709,A -85,B 0,C 180,E1 -19694.98,E2 -19694.98} C_VEL
LIN {X 0,Y 355.849,Z 383.015,A -85,B 0,C 180,E1 -19696.652,E2 -19696.652} C_VEL
LIN {X 0,Y 359.401,Z 385.211,A -85,B 0,C 180,E1 -19697.884,E2 -19697.884} C_VEL
LIN {X 0,Y 363.782,Z 388.487,A -85,B 0,C 180,E1 -19699.69,E2 -19699.69} C_VEL
LIN {X 0,Y 366.921,Z 390.493,A -85,B 0,C 180,E1 -19701.186,E2 -19701.186} C_VEL
LIN {X 0,Y 369.068,Z 391.655,A -85,B 0,C 180,E1 -19702.34,E2 -19702.34} C_VEL
LIN {X 0,Y 370.864,Z 392.574,A -85,B 0,C 180,E1 -19703.471,E2 -19703.471} C_VEL
LIN {X 0,Y 372.383,Z 393.232,A -85,B 0,C 180,E1 -19704.585,E2 -19704.585} C_VEL
LIN {X 0,Y 373.639,Z 393.667,A -85,B 0,C 180,E1 -19705.685,E2 -19705.685} C_VEL
LIN {X 0,Y 374.62,Z 393.933,A -85,B 0,C 180,E1 -19706.774,E2 -19706.774} C_VEL
LIN {X 0,Y 375.246,Z 394.328,A -85,B 0,C 180,E1 -19707.853,E2 -19707.853} C_VEL
LIN {X 0,Y 375.608,Z 394.598,A -85,B 0,C 180,E1 -19708.928,E2 -19708.928} C_VEL
LIN {X 0,Y 375.784,Z 394.512,A -85,B 0,C 180,E1 -19710,E2 -19710} C_VEL
LIN {X 0,Y 375.629,Z 394.538,A -85,B 0,C 180,E1 -19711.072,E2 -19711.072} C_VEL
LIN {X 0,Y 375.268,Z 394.277,A -85,B 0,C 180,E1 -19712.147,E2 -19712.147} C_VEL
LIN {X 0,Y 374.624,Z 393.951,A -85,B 0,C 180,E1 -19713.226,E2 -19713.226} C_VEL
LIN {X 0,Y 373.577,Z 393.66,A -85,B 0,C 180,E1 -19714.394,E2 -19714.394} C_VEL
LIN {X 0,Y 372.396,Z 393.264,A -85,B 0,C 180,E1 -19715.415,E2 -19715.415} C_VEL
LIN {X 0,Y 370.877,Z 392.593,A -85,B 0,C 180,E1 -19716.529,E2 -19716.529} C_VEL
LIN {X 0,Y 368.834,Z 391.579,A -85,B 0,C 180,E1 -19717.767,E2 -19717.767} C_VEL
LIN {X 0,Y 365.355,Z 389.551,A -85,B 0,C 180,E1 -19719.585,E2 -19719.585} C_VEL
LIN {X 0,Y 361.062,Z 386.518,A -85,B 0,C 180,E1 -19721.453,E2 -19721.453} C_VEL
LIN {X 0,Y 357.702,Z 384.026,A -85,B 0,C 180,E1 -19722.733,E2 -19722.733} C_VEL
LIN {X 0,Y 352.111,Z 380.804,A -85,B 0,C 180,E1 -19724.511,E2 -19724.511} C_VEL
LIN {X 0,Y 345.815,Z 376.516,A -85,B 0,C 180,E1 -19726.287,E2 -19726.287} C_VEL
LIN {X 0,Y 340.187,Z 372.425,A -85,B 0,C 180,E1 -19727.715,E2 -19727.715} C_VEL
LIN {X 0,Y 332.642,Z 367.152,A -85,B 0,C 180,E1 -19729.415,E2 -19729.415} C_VEL
LIN {X 0,Y 326.059,Z 362.178,A -85,B 0,C 180,E1 -19730.752,E2 -19730.752} C_VEL
LIN {X 0,Y 318.316,Z 356.304,A -85,B 0,C 180,E1 -19732.158,E2 -19732.158} C_VEL
LIN {X 0,Y 310.344,Z 350.167,A -85,B 0,C 180,E1 -19733.386,E2 -19733.386} C_VEL
LIN {X 0,Y 302.137,Z 343.351,A -85,B 0,C 180,E1 -19734.485,E2 -19734.485} C_VEL
LIN {X 0,Y 289.331,Z 332.268,A -85,B 0,C 180,E1 -19736.008,E2 -19736.008} C_VEL
LIN {X 0,Y 274.584,Z 317.2,A -85,B 0,C 180,E1 -19737.969,E2 -19737.969} C_VEL
LIN {X 0,Y 265.406,Z 306.053,A -85,B 0,C 180,E1 -19739.375,E2 -19739.375} C_VEL
LIN {X 0,Y 256.871,Z 293.463,A -85,B 0,C 180,E1 -19740.862,E2 -19740.862} C_VEL
LIN {X 0,Y 247.788,Z 276.053,A -85,B 0,C 180,E1 -19742.722,E2 -19742.722} C_VEL
LIN {X 0,Y 238.791,Z 260.042,A -85,B 0,C 180,E1 -19744.704,E2 -19744.704} C_VEL
LIN {X 0,Y 236.394,Z 256.108,A -85,B 0,C 180,E1 -19745.253,E2 -19745.253} C_VEL
LIN {X 0,Y 235.131,Z 253.431,A -85,B 0,C 180,E1 -19745.648,E2 -19745.648} C_VEL
LIN {X 0,Y 234.953,Z 252.731,A -85,B 0,C 180,E1 -19746.136,E2 -19746.136} C_VEL
LIN {X 0,Y 234.938,Z 252.698,A -85,B 0,C 180,E1 -19748.945,E2 -19748.945} C_VEL
LIN {X 0,Y 234.894,Z 252.67,A -85,B 0,C 180,E1 -19753.484,E2 -19753.484} C_VEL
LIN {X 0,Y 234.962,Z 252.719,A -85,B 0,C 180,E1 -19756.533,E2 -19756.533} C_VEL
LIN {X 0,Y 234.952,Z 252.711,A -85,B 0,C 180,E1 -19761.087,E2 -19761.087} C_VEL
LIN {X 0,Y 234.958,Z 252.692,A -85,B 0,C 180,E1 -19765.368,E2 -19765.368} C_VEL
LIN {X 0,Y 234.921,Z 252.723,A -85,B 0,C 180,E1 -19769.432,E2 -19769.432} C_VEL
LIN {X 0,Y 234.991,Z 252.684,A -85,B 0,C 180,E1 -19773.795,E2 -19773.795} C_VEL
LIN {X 0,Y 234.996,Z 252.688,A -85,B 0,C 180,E1 -19778.969,E2 -19778.969} C_VEL
LIN {X 0,Y 235.095,Z 252.68,A -85,B 0,C 180,E1 -19783.061,E2 -19783.061} C_VEL
LIN {X 0,Y 235.114,Z 252.672,A -85,B 0,C 180,E1 -19787.923,E2 -19787.923} C_VEL
LIN {X 0,Y 235.33,Z 252.633,A -85,B 0,C 180,E1 -19791.413,E2 -19791.413} C_VEL
LIN {X 0,Y 235.392,Z 252.653,A -85,B 0,C 180,E1 -19793.142,E2 -19793.142} C_VEL
LIN {X 0,Y 235.595,Z 252.6,A -85,B 0,C 180,E1 -19798.292,E2 -19798.292} C_VEL
LIN {X 0,Y 235.595,Z 252.607,A -85,B 0,C 180,E1 -19801.71,E2 -19801.71} C_VEL
LIN {X 0,Y 235.354,Z 252.651,A -85,B 0,C 180,E1 -19806.861,E2 -19806.861} C_VEL
LIN {X 0,Y 235.214,Z 252.641,A -85,B 0,C 180,E1 -19810.328,E2 -19810.328} C_VEL
LIN {X 0,Y 235.081,Z 252.693,A -85,B 0,C 180,E1 -19815.61,E2 -19815.61} C_VEL
LIN {X 0,Y 234.998,Z 252.671,A -85,B 0,C 180,E1 -19819.207,E2 -19819.207} C_VEL
LIN {X 0,Y 234.962,Z 252.716,A -85,B 0,C 180,E1 -19822.884,E2 -19822.884} C_VEL
LIN {X 0,Y 234.969,Z 252.682,A -85,B 0,C 180,E1 -19826.658,E2 -19826.658} C_VEL
LIN {X 0,Y 234.924,Z 252.723,A -85,B 0,C 180,E1 -19830.57,E2 -19830.57} C_VEL
LIN {X 0,Y 234.935,Z 252.694,A -85,B 0,C 180,E1 -19834.638,E2 -19834.638} C_VEL
LIN {X 0,Y 234.944,Z 252.706,A -85,B 0,C 180,E1 -19838.945,E2 -19838.945} C_VEL
LIN {X 0,Y 234.882,Z 252.72,A -85,B 0,C 180,E1 -19843.488,E2 -19843.488} C_VEL
LIN {X 0,Y 234.893,Z 252.7,A -85,B 0,C 180,E1 -19848.056,E2 -19848.056} C_VEL
LIN {X 0,Y 234.933,Z 252.901,A -85,B 0,C 180,E1 -19848.569,E2 -19848.569} C_VEL
LIN {X 0,Y 236.481,Z 259.233,A -85,B 0,C 180,E1 -19852.43,E2 -19852.43} C_VEL
LIN {X 0,Y 237.32,Z 263.397,A -85,B 0,C 180,E1 -19854.703,E2 -19854.703} C_VEL
LIN {X 0,Y 239.062,Z 267.24,A -85,B 0,C 180,E1 -19855.217,E2 -19855.217} C_VEL
LIN {X 0,Y 246.785,Z 284.02,A -85,B 0,C 180,E1 -19857.016,E2 -19857.016} C_VEL
LIN {X 0,Y 249.462,Z 290.811,A -85,B 0,C 180,E1 -19857.637,E2 -19857.637} C_VEL
LIN {X 0,Y 250.343,Z 296.466,A -85,B 0,C 180,E1 -19857.952,E2 -19857.952} C_VEL
LIN {X 0,Y 250.292,Z 302.334,A -85,B 0,C 180,E1 -19858.138,E2 -19858.138} C_VEL
LIN {X 0,Y 248.041,Z 322.266,A -85,B 0,C 180,E1 -19858.481,E2 -19858.481} C_VEL
LIN {X 0,Y 246.193,Z 369.865,A -85,B 0,C 180,E1 -19859.863,E2 -19859.863} C_VEL
LIN {X 0,Y 245.234,Z 380.707,A -85,B 0,C 180,E1 -19860.369,E2 -19860.369} C_VEL
LIN {X 0,Y 243.659,Z 393.259,A -85,B 0,C 180,E1 -19861.228,E2 -19861.228} C_VEL
LIN {X 0,Y 241.475,Z 405.969,A -85,B 0,C 180,E1 -19862.482,E2 -19862.482} C_VEL
LIN {X 0,Y 239.642,Z 415.242,A -85,B 0,C 180,E1 -19863.668,E2 -19863.668} C_VEL
LIN {X 0,Y 237.681,Z 424.186,A -85,B 0,C 180,E1 -19865.08,E2 -19865.08} C_VEL
LIN {X 0,Y 235.514,Z 432.709,A -85,B 0,C 180,E1 -19866.71,E2 -19866.71} C_VEL
LIN {X 0,Y 233.657,Z 439.927,A -85,B 0,C 180,E1 -19868.379,E2 -19868.379} C_VEL
LIN {X 0,Y 232.042,Z 446.462,A -85,B 0,C 180,E1 -19870.189,E2 -19870.189} C_VEL
LIN {X 0,Y 230.267,Z 452.666,A -85,B 0,C 180,E1 -19872.229,E2 -19872.229} C_VEL
LIN {X 0,Y 229.074,Z 457.169,A -85,B 0,C 180,E1 -19873.971,E2 -19873.971} C_VEL
LIN {X 0,Y 227.548,Z 462.66,A -85,B 0,C 180,E1 -19876.606,E2 -19876.606} C_VEL
LIN {X 0,Y 226.575,Z 466.99,A -85,B 0,C 180,E1 -19879.274,E2 -19879.274} C_VEL
LIN {X 0,Y 226.135,Z 469.36,A -85,B 0,C 180,E1 -19881.06,E2 -19881.06} C_VEL
LIN {X 0,Y 225.811,Z 471.162,A -85,B 0,C 180,E1 -19882.849,E2 -19882.849} C_VEL
LIN {X 0,Y 225.588,Z 473.616,A -85,B 0,C 180,E1 -19886.428,E2 -19886.428} C_VEL
LIN {X 0,Y 225.625,Z 474.209,A -85,B 0,C 180,E1 -19888.215,E2 -19888.215} C_VEL
LIN {X 0,Y 225.708,Z 474.366,A -85,B 0,C 180,E1 -19890,E2 -19890} C_VEL
LIN {X 0,Y 225.624,Z 474.209,A -85,B 0,C 180,E1 -19891.785,E2 -19891.785} C_VEL
LIN {X 0,Y 225.587,Z 473.142,A -85,B 0,C 180,E1 -19894.475,E2 -19894.475} C_VEL
LIN {X 0,Y 225.778,Z 471.161,A -85,B 0,C 180,E1 -19897.153,E2 -19897.153} C_VEL
LIN {X 0,Y 226.328,Z 468.208,A -85,B 0,C 180,E1 -19899.834,E2 -19899.834} C_VEL
LIN {X 0,Y 227.203,Z 464.216,A -85,B 0,C 180,E1 -19902.505,E2 -19902.505} C_VEL
LIN {X 0,Y 228.51,Z 459.084,A -85,B 0,C 180,E1 -19905.155,E2 -19905.155} C_VEL
LIN {X 0,Y 229.976,Z 453.823,A -85,B 0,C 180,E1 -19907.335,E2 -19907.335} C_VEL
LIN {X 0,Y 231.748,Z 447.508,A -85,B 0,C 180,E1 -19909.486,E2 -19909.486} C_VEL
LIN {X 0,Y 233.277,Z 441.555,A -85,B 0,C 180,E1 -19911.194,E2 -19911.194} C_VEL
LIN {X 0,Y 235.03,Z 434.628,A -85,B 0,C 180,E1 -19912.876,E2 -19912.876} C_VEL
LIN {X 0,Y 237.119,Z 426.453,A -85,B 0,C 180,E1 -19914.516,E2 -19914.516} C_VEL
LIN {X 0,Y 239.08,Z 417.945,A -85,B 0,C 180,E1 -19915.929,E2 -19915.929} C_VEL
LIN {X 0,Y 240.854,Z 409.232,A -85,B 0,C 180,E1 -19917.125,E2 -19917.125} C_VEL
LIN {X 0,Y 242.464,Z 400.484,A -85,B 0,C 180,E1 -19918.1,E2 -19918.1} C_VEL
LIN {X 0,Y 244.02,Z 390.687,A -85,B 0,C 180,E1 -19918.961,E2 -19918.961} C_VEL
LIN {X 0,Y 245.223,Z 380.713,A -85,B 0,C 180,E1 -19919.632,E2 -19919.632} C_VEL
LIN {X 0,Y 246.111,Z 371.043,A -85,B 0,C 180,E1 -19920.094,E2 -19920.094} C_VEL
LIN {X 0,Y 247.083,Z 348.083,A -85,B 0,C 180,E1 -19920.796,E2 -19920.796} C_VEL
LIN {X 0,Y 248.13,Z 318.678,A -85,B 0,C 180,E1 -19921.625,E2 -19921.625} C_VEL
LIN {X 0,Y 244.5,Z 297.403,A -85,B 0,C 180,E1 -19922.871,E2 -19922.871} C_VEL
LIN {X 0,Y 243.267,Z 292.05,A -85,B 0,C 180,E1 -19923.242,E2 -19923.242} C_VEL
LIN {X 0,Y 235.996,Z 275.468,A -85,B 0,C 180,E1 -19924.998,E2 -19924.998} C_VEL
LIN {X 0,Y 230.183,Z 263.511,A -85,B 0,C 180,E1 -19926.503,E2 -19926.503} C_VEL
